; ----- Contour 2 -----
PTP {X 107.78, Y 86.02, Z 10.00, A 0, B 0, C 0}
LIN {X 107.78, Y 86.02, Z 0.00, A 0, B 0, C 0}
LIN {X 107.56, Y 86.02, Z 0.00, A 0, B 0, C 0} C_DIS
LIN {X 107.34, Y 86.02, Z 0.00, A 0, B 0, C 0} C_DIS
LIN {X 107.12, Y 86.02, Z 0.00, A 0, B 0, C 0} C_DIS
LIN {X 106.90, Y 86.02, Z 0.00, A 0, B 0, C 0} C_DIS
LIN {X 106.69, Y 86.03, Z 0.00, A 0, B 0, C 0} C_DIS
LIN {X 106.47, Y 86.03, Z 0.00, A 0, B 0, C 0} C_DIS
LIN {X 106.25, Y 86.04, Z 0.00, A 0, B 0, C 0} C_DIS
LIN {X 106.03, Y 86.04, Z 0.00, A 0, B 0, C 0} C_DIS
LIN {X 105.82, Y 86.04, Z 0.00, A 0, B 0, C 0} C_DIS
LIN {X 105.60, Y 86.03, Z 0.00, A 0, B 0, C 0} C_DIS
LIN {X 105.38, Y 86.02, Z 0.00, A 0, B 0, C 0} C_DIS
LIN {X 105.17, Y 86.00, Z 0.00, A 0, B 0, C 0} C_DIS
LIN {X 104.95, Y 85.97, Z 0.00, A 0, B 0, C 0} C_DIS
LIN {X 104.74, Y 85.94, Z 0.00, A 0, B 0, C 0} C_DIS
LIN {X 104.52, Y 85.90, Z 0.00, A 0, B 0, C 0} C_DIS
LIN {X 104.31, Y 85.85, Z 0.00, A 0, B 0, C 0} C_DIS
LIN {X 104.09, Y 85.79, Z 0.00, A 0, B 0, C 0} C_DIS
LIN {X 103.88, Y 85.73, Z 0.00, A 0, B 0, C 0} C_DIS
LIN {X 103.67, Y 85.67, Z 0.00, A 0, B 0, C 0} C_DIS
LIN {X 103.45, Y 85.60, Z 0.00, A 0, B 0, C 0} C_DIS
LIN {X 103.24, Y 85.53, Z 0.00, A 0, B 0, C 0} C_DIS
LIN {X 103.03, Y 85.46, Z 0.00, A 0, B 0, C 0} C_DIS
LIN {X 102.82, Y 85.39, Z 0.00, A 0, B 0, C 0} C_DIS
LIN {X 102.61, Y 85.31, Z 0.00, A 0, B 0, C 0} C_DIS
LIN {X 102.40, Y 85.24, Z 0.00, A 0, B 0, C 0} C_DIS
LIN {X 102.18, Y 85.17, Z 0.00, A 0, B 0, C 0} C_DIS
LIN {X 101.97, Y 85.09, Z 0.00, A 0, B 0, C 0} C_DIS
LIN {X 101.76, Y 85.01, Z 0.00, A 0, B 0, C 0} C_DIS
LIN {X 101.55, Y 84.94, Z 0.00, A 0, B 0, C 0} C_DIS
LIN {X 101.34, Y 84.85, Z 0.00, A 0, B 0, C 0} C_DIS
LIN {X 101.14, Y 84.77, Z 0.00, A 0, B 0, C 0} C_DIS
LIN {X 100.93, Y 84.68, Z 0.00, A 0, B 0, C 0} C_DIS
LIN {X 100.72, Y 84.58, Z 0.00, A 0, B 0, C 0} C_DIS
LIN {X 100.51, Y 84.48, Z 0.00, A 0, B 0, C 0} C_DIS
LIN {X 100.31, Y 84.38, Z 0.00, A 0, B 0, C 0} C_DIS
LIN {X 100.10, Y 84.27, Z 0.00, A 0, B 0, C 0} C_DIS
LIN {X 99.90, Y 84.15, Z 0.00, A 0, B 0, C 0} C_DIS
LIN {X 99.70, Y 84.02, Z 0.00, A 0, B 0, C 0} C_DIS
LIN {X 99.50, Y 83.89, Z 0.00, A 0, B 0, C 0} C_DIS
LIN {X 99.31, Y 83.74, Z 0.00, A 0, B 0, C 0} C_DIS
LIN {X 99.11, Y 83.59, Z 0.00, A 0, B 0, C 0} C_DIS
LIN {X 98.93, Y 83.43, Z 0.00, A 0, B 0, C 0} C_DIS
LIN {X 98.74, Y 83.26, Z 0.00, A 0, B 0, C 0} C_DIS
LIN {X 98.56, Y 83.08, Z 0.00, A 0, B 0, C 0} C_DIS
LIN {X 98.38, Y 82.89, Z 0.00, A 0, B 0, C 0} C_DIS
LIN {X 98.20, Y 82.72, Z 0.00, A 0, B 0, C 0} C_DIS
LIN {X 98.01, Y 82.56, Z 0.00, A 0, B 0, C 0} C_DIS
LIN {X 97.82, Y 82.41, Z 0.00, A 0, B 0, C 0} C_DIS
LIN {X 97.62, Y 82.28, Z 0.00, A 0, B 0, C 0} C_DIS
LIN {X 97.42, Y 82.13, Z 0.00, A 0, B 0, C 0} C_DIS
LIN {X 97.23, Y 81.97, Z 0.00, A 0, B 0, C 0} C_DIS
LIN {X 97.05, Y 81.80, Z 0.00, A 0, B 0, C 0} C_DIS
LIN {X 96.87, Y 81.61, Z 0.00, A 0, B 0, C 0} C_DIS
LIN {X 96.71, Y 81.40, Z 0.00, A 0, B 0, C 0} C_DIS
LIN {X 96.55, Y 81.17, Z 0.00, A 0, B 0, C 0} C_DIS
LIN {X 96.40, Y 80.93, Z 0.00, A 0, B 0, C 0} C_DIS
LIN {X 96.26, Y 80.69, Z 0.00, A 0, B 0, C 0} C_DIS
LIN {X 96.10, Y 80.45, Z 0.00, A 0, B 0, C 0} C_DIS
LIN {X 95.94, Y 80.23, Z 0.00, A 0, B 0, C 0} C_DIS
LIN {X 95.78, Y 80.01, Z 0.00, A 0, B 0, C 0} C_DIS
LIN {X 95.61, Y 79.81, Z 0.00, A 0, B 0, C 0} C_DIS
LIN {X 95.44, Y 79.60, Z 0.00, A 0, B 0, C 0} C_DIS
LIN {X 95.28, Y 79.39, Z 0.00, A 0, B 0, C 0} C_DIS
LIN {X 95.11, Y 79.18, Z 0.00, A 0, B 0, C 0} C_DIS
LIN {X 94.95, Y 78.96, Z 0.00, A 0, B 0, C 0} C_DIS
LIN {X 94.80, Y 78.73, Z 0.00, A 0, B 0, C 0} C_DIS
LIN {X 94.64, Y 78.51, Z 0.00, A 0, B 0, C 0} C_DIS
LIN {X 94.49, Y 78.27, Z 0.00, A 0, B 0, C 0} C_DIS
LIN {X 94.34, Y 78.04, Z 0.00, A 0, B 0, C 0} C_DIS
LIN {X 94.20, Y 77.80, Z 0.00, A 0, B 0, C 0} C_DIS
LIN {X 94.06, Y 77.55, Z 0.00, A 0, B 0, C 0} C_DIS
LIN {X 93.92, Y 77.31, Z 0.00, A 0, B 0, C 0} C_DIS
LIN {X 93.78, Y 77.05, Z 0.00, A 0, B 0, C 0} C_DIS
LIN {X 93.64, Y 76.80, Z 0.00, A 0, B 0, C 0} C_DIS
LIN {X 93.51, Y 76.54, Z 0.00, A 0, B 0, C 0} C_DIS
LIN {X 93.38, Y 76.28, Z 0.00, A 0, B 0, C 0} C_DIS
LIN {X 93.25, Y 76.01, Z 0.00, A 0, B 0, C 0} C_DIS
LIN {X 93.13, Y 75.74, Z 0.00, A 0, B 0, C 0} C_DIS
LIN {X 93.00, Y 75.47, Z 0.00, A 0, B 0, C 0} C_DIS
LIN {X 92.88, Y 75.20, Z 0.00, A 0, B 0, C 0} C_DIS
LIN {X 92.76, Y 74.93, Z 0.00, A 0, B 0, C 0} C_DIS
LIN {X 92.64, Y 74.65, Z 0.00, A 0, B 0, C 0} C_DIS
LIN {X 92.53, Y 74.38, Z 0.00, A 0, B 0, C 0} C_DIS
LIN {X 92.41, Y 74.10, Z 0.00, A 0, B 0, C 0} C_DIS
LIN {X 92.30, Y 73.82, Z 0.00, A 0, B 0, C 0} C_DIS
LIN {X 92.19, Y 73.54, Z 0.00, A 0, B 0, C 0} C_DIS
LIN {X 92.08, Y 73.26, Z 0.00, A 0, B 0, C 0} C_DIS
LIN {X 91.98, Y 72.97, Z 0.00, A 0, B 0, C 0} C_DIS
LIN {X 91.87, Y 72.69, Z 0.00, A 0, B 0, C 0} C_DIS
LIN {X 91.77, Y 72.40, Z 0.00, A 0, B 0, C 0} C_DIS
LIN {X 91.67, Y 72.11, Z 0.00, A 0, B 0, C 0} C_DIS
LIN {X 91.57, Y 71.82, Z 0.00, A 0, B 0, C 0} C_DIS
LIN {X 91.48, Y 71.52, Z 0.00, A 0, B 0, C 0} C_DIS
LIN {X 91.39, Y 71.23, Z 0.00, A 0, B 0, C 0} C_DIS
LIN {X 91.30, Y 70.93, Z 0.00, A 0, B 0, C 0} C_DIS
LIN {X 91.22, Y 70.63, Z 0.00, A 0, B 0, C 0} C_DIS
LIN {X 91.14, Y 70.32, Z 0.00, A 0, B 0, C 0} C_DIS
LIN {X 91.06, Y 70.02, Z 0.00, A 0, B 0, C 0} C_DIS
LIN {X 91.00, Y 69.71, Z 0.00, A 0, B 0, C 0} C_DIS
LIN {X 90.94, Y 69.39, Z 0.00, A 0, B 0, C 0} C_DIS
LIN {X 90.88, Y 69.08, Z 0.00, A 0, B 0, C 0} C_DIS
LIN {X 90.83, Y 68.76, Z 0.00, A 0, B 0, C 0} C_DIS
LIN {X 90.79, Y 68.44, Z 0.00, A 0, B 0, C 0} C_DIS
LIN {X 90.74, Y 68.12, Z 0.00, A 0, B 0, C 0} C_DIS
LIN {X 90.69, Y 67.80, Z 0.00, A 0, B 0, C 0} C_DIS
LIN {X 90.63, Y 67.48, Z 0.00, A 0, B 0, C 0} C_DIS
LIN {X 90.57, Y 67.17, Z 0.00, A 0, B 0, C 0} C_DIS
LIN {X 90.50, Y 66.86, Z 0.00, A 0, B 0, C 0} C_DIS
LIN {X 90.42, Y 66.56, Z 0.00, A 0, B 0, C 0} C_DIS
LIN {X 90.34, Y 66.25, Z 0.00, A 0, B 0, C 0} C_DIS
LIN {X 90.26, Y 65.94, Z 0.00, A 0, B 0, C 0} C_DIS
LIN {X 90.20, Y 65.63, Z 0.00, A 0, B 0, C 0} C_DIS
LIN {X 90.15, Y 65.31, Z 0.00, A 0, B 0, C 0} C_DIS
LIN {X 90.11, Y 64.99, Z 0.00, A 0, B 0, C 0} C_DIS
LIN {X 90.08, Y 64.67, Z 0.00, A 0, B 0, C 0} C_DIS
LIN {X 90.05, Y 64.34, Z 0.00, A 0, B 0, C 0} C_DIS
LIN {X 90.04, Y 64.01, Z 0.00, A 0, B 0, C 0} C_DIS
LIN {X 90.03, Y 63.69, Z 0.00, A 0, B 0, C 0} C_DIS
LIN {X 90.02, Y 63.36, Z 0.00, A 0, B 0, C 0} C_DIS
LIN {X 90.02, Y 63.03, Z 0.00, A 0, B 0, C 0} C_DIS
LIN {X 90.02, Y 62.70, Z 0.00, A 0, B 0, C 0} C_DIS
LIN {X 90.02, Y 62.38, Z 0.00, A 0, B 0, C 0} C_DIS
LIN {X 90.03, Y 62.05, Z 0.00, A 0, B 0, C 0} C_DIS
LIN {X 90.03, Y 61.72, Z 0.00, A 0, B 0, C 0} C_DIS
LIN {X 90.03, Y 61.39, Z 0.00, A 0, B 0, C 0} C_DIS
LIN {X 90.03, Y 61.07, Z 0.00, A 0, B 0, C 0} C_DIS
LIN {X 90.03, Y 60.74, Z 0.00, A 0, B 0, C 0} C_DIS
LIN {X 90.03, Y 60.41, Z 0.00, A 0, B 0, C 0} C_DIS
LIN {X 90.03, Y 60.08, Z 0.00, A 0, B 0, C 0} C_DIS
LIN {X 90.03, Y 59.76, Z 0.00, A 0, B 0, C 0} C_DIS
LIN {X 90.03, Y 59.43, Z 0.00, A 0, B 0, C 0} C_DIS
LIN {X 90.03, Y 59.10, Z 0.00, A 0, B 0, C 0} C_DIS
LIN {X 90.03, Y 58.77, Z 0.00, A 0, B 0, C 0} C_DIS
LIN {X 90.03, Y 58.44, Z 0.00, A 0, B 0, C 0} C_DIS
LIN {X 90.03, Y 58.12, Z 0.00, A 0, B 0, C 0} C_DIS
LIN {X 90.03, Y 57.79, Z 0.00, A 0, B 0, C 0} C_DIS
LIN {X 90.03, Y 57.46, Z 0.00, A 0, B 0, C 0} C_DIS
LIN {X 90.03, Y 57.13, Z 0.00, A 0, B 0, C 0} C_DIS
LIN {X 90.03, Y 56.80, Z 0.00, A 0, B 0, C 0} C_DIS
LIN {X 90.03, Y 56.48, Z 0.00, A 0, B 0, C 0} C_DIS
LIN {X 90.03, Y 56.15, Z 0.00, A 0, B 0, C 0} C_DIS
LIN {X 90.03, Y 55.82, Z 0.00, A 0, B 0, C 0} C_DIS
LIN {X 90.03, Y 55.49, Z 0.00, A 0, B 0, C 0} C_DIS
LIN {X 90.03, Y 55.17, Z 0.00, A 0, B 0, C 0} C_DIS
LIN {X 90.03, Y 54.84, Z 0.00, A 0, B 0, C 0} C_DIS
LIN {X 90.03, Y 54.51, Z 0.00, A 0, B 0, C 0} C_DIS
LIN {X 90.03, Y 54.18, Z 0.00, A 0, B 0, C 0} C_DIS
LIN {X 90.03, Y 53.86, Z 0.00, A 0, B 0, C 0} C_DIS
LIN {X 90.03, Y 53.53, Z 0.00, A 0, B 0, C 0} C_DIS
LIN {X 90.03, Y 53.20, Z 0.00, A 0, B 0, C 0} C_DIS
LIN {X 90.03, Y 52.87, Z 0.00, A 0, B 0, C 0} C_DIS
LIN {X 90.03, Y 52.55, Z 0.00, A 0, B 0, C 0} C_DIS
LIN {X 90.03, Y 52.22, Z 0.00, A 0, B 0, C 0} C_DIS
LIN {X 90.03, Y 51.89, Z 0.00, A 0, B 0, C 0} C_DIS
LIN {X 90.03, Y 51.56, Z 0.00, A 0, B 0, C 0} C_DIS
LIN {X 90.03, Y 51.24, Z 0.00, A 0, B 0, C 0} C_DIS
LIN {X 90.03, Y 50.91, Z 0.00, A 0, B 0, C 0} C_DIS
LIN {X 90.03, Y 50.58, Z 0.00, A 0, B 0, C 0} C_DIS
LIN {X 90.03, Y 50.25, Z 0.00, A 0, B 0, C 0} C_DIS
LIN {X 90.03, Y 49.92, Z 0.00, A 0, B 0, C 0} C_DIS
LIN {X 90.03, Y 49.60, Z 0.00, A 0, B 0, C 0} C_DIS
LIN {X 90.02, Y 49.27, Z 0.00, A 0, B 0, C 0} C_DIS
LIN {X 90.02, Y 48.94, Z 0.00, A 0, B 0, C 0} C_DIS
LIN {X 90.02, Y 48.61, Z 0.00, A 0, B 0, C 0} C_DIS
LIN {X 90.02, Y 48.28, Z 0.00, A 0, B 0, C 0} C_DIS
LIN {X 90.02, Y 47.95, Z 0.00, A 0, B 0, C 0} C_DIS
LIN {X 90.03, Y 47.62, Z 0.00, A 0, B 0, C 0} C_DIS
LIN {X 90.04, Y 47.30, Z 0.00, A 0, B 0, C 0} C_DIS
LIN {X 90.06, Y 46.97, Z 0.00, A 0, B 0, C 0} C_DIS
LIN {X 90.08, Y 46.65, Z 0.00, A 0, B 0, C 0} C_DIS
LIN {X 90.11, Y 46.33, Z 0.00, A 0, B 0, C 0} C_DIS
LIN {X 90.15, Y 46.01, Z 0.00, A 0, B 0, C 0} C_DIS
LIN {X 90.19, Y 45.69, Z 0.00, A 0, B 0, C 0} C_DIS
LIN {X 90.24, Y 45.37, Z 0.00, A 0, B 0, C 0} C_DIS
LIN {X 90.30, Y 45.06, Z 0.00, A 0, B 0, C 0} C_DIS
LIN {X 90.37, Y 44.75, Z 0.00, A 0, B 0, C 0} C_DIS
LIN {X 90.44, Y 44.44, Z 0.00, A 0, B 0, C 0} C_DIS
LIN {X 90.52, Y 44.13, Z 0.00, A 0, B 0, C 0} C_DIS
LIN {X 90.60, Y 43.83, Z 0.00, A 0, B 0, C 0} C_DIS
LIN {X 90.69, Y 43.53, Z 0.00, A 0, B 0, C 0} C_DIS
LIN {X 90.78, Y 43.23, Z 0.00, A 0, B 0, C 0} C_DIS
LIN {X 90.87, Y 42.93, Z 0.00, A 0, B 0, C 0} C_DIS
LIN {X 90.96, Y 42.63, Z 0.00, A 0, B 0, C 0} C_DIS
LIN {X 91.05, Y 42.34, Z 0.00, A 0, B 0, C 0} C_DIS
LIN {X 91.15, Y 42.04, Z 0.00, A 0, B 0, C 0} C_DIS
LIN {X 91.24, Y 41.75, Z 0.00, A 0, B 0, C 0} C_DIS
LIN {X 91.34, Y 41.46, Z 0.00, A 0, B 0, C 0} C_DIS
LIN {X 91.44, Y 41.17, Z 0.00, A 0, B 0, C 0} C_DIS
LIN {X 91.54, Y 40.89, Z 0.00, A 0, B 0, C 0} C_DIS
LIN {X 91.64, Y 40.60, Z 0.00, A 0, B 0, C 0} C_DIS
LIN {X 91.75, Y 40.32, Z 0.00, A 0, B 0, C 0} C_DIS
LIN {X 91.85, Y 40.03, Z 0.00, A 0, B 0, C 0} C_DIS
LIN {X 91.96, Y 39.75, Z 0.00, A 0, B 0, C 0} C_DIS
LIN {X 92.08, Y 39.47, Z 0.00, A 0, B 0, C 0} C_DIS
LIN {X 92.19, Y 39.19, Z 0.00, A 0, B 0, C 0} C_DIS
LIN {X 92.31, Y 38.92, Z 0.00, A 0, B 0, C 0} C_DIS
LIN {X 92.43, Y 38.64, Z 0.00, A 0, B 0, C 0} C_DIS
LIN {X 92.55, Y 38.37, Z 0.00, A 0, B 0, C 0} C_DIS
LIN {X 92.68, Y 38.11, Z 0.00, A 0, B 0, C 0} C_DIS
LIN {X 92.81, Y 37.84, Z 0.00, A 0, B 0, C 0} C_DIS
LIN {X 92.94, Y 37.59, Z 0.00, A 0, B 0, C 0} C_DIS
LIN {X 93.08, Y 37.33, Z 0.00, A 0, B 0, C 0} C_DIS
LIN {X 93.22, Y 37.08, Z 0.00, A 0, B 0, C 0} C_DIS
LIN {X 93.37, Y 36.84, Z 0.00, A 0, B 0, C 0} C_DIS
LIN {X 93.51, Y 36.60, Z 0.00, A 0, B 0, C 0} C_DIS
LIN {X 93.66, Y 36.36, Z 0.00, A 0, B 0, C 0} C_DIS
LIN {X 93.81, Y 36.12, Z 0.00, A 0, B 0, C 0} C_DIS
LIN {X 93.97, Y 35.89, Z 0.00, A 0, B 0, C 0} C_DIS
LIN {X 94.12, Y 35.66, Z 0.00, A 0, B 0, C 0} C_DIS
LIN {X 94.27, Y 35.43, Z 0.00, A 0, B 0, C 0} C_DIS
LIN {X 94.43, Y 35.20, Z 0.00, A 0, B 0, C 0} C_DIS
LIN {X 94.58, Y 34.97, Z 0.00, A 0, B 0, C 0} C_DIS
LIN {X 94.74, Y 34.74, Z 0.00, A 0, B 0, C 0} C_DIS
LIN {X 94.89, Y 34.51, Z 0.00, A 0, B 0, C 0} C_DIS
LIN {X 95.05, Y 34.28, Z 0.00, A 0, B 0, C 0} C_DIS
LIN {X 95.20, Y 34.05, Z 0.00, A 0, B 0, C 0} C_DIS
LIN {X 95.35, Y 33.82, Z 0.00, A 0, B 0, C 0} C_DIS
LIN {X 95.51, Y 33.58, Z 0.00, A 0, B 0, C 0} C_DIS
LIN {X 95.66, Y 33.35, Z 0.00, A 0, B 0, C 0} C_DIS
LIN {X 95.82, Y 33.12, Z 0.00, A 0, B 0, C 0} C_DIS
LIN {X 95.97, Y 32.89, Z 0.00, A 0, B 0, C 0} C_DIS
LIN {X 96.13, Y 32.66, Z 0.00, A 0, B 0, C 0} C_DIS
LIN {X 96.28, Y 32.43, Z 0.00, A 0, B 0, C 0} C_DIS
LIN {X 96.43, Y 32.20, Z 0.00, A 0, B 0, C 0} C_DIS
LIN {X 96.59, Y 31.97, Z 0.00, A 0, B 0, C 0} C_DIS
LIN {X 96.74, Y 31.73, Z 0.00, A 0, B 0, C 0} C_DIS
LIN {X 96.90, Y 31.50, Z 0.00, A 0, B 0, C 0} C_DIS
LIN {X 97.05, Y 31.27, Z 0.00, A 0, B 0, C 0} C_DIS
LIN {X 97.20, Y 31.04, Z 0.00, A 0, B 0, C 0} C_DIS
LIN {X 97.36, Y 30.81, Z 0.00, A 0, B 0, C 0} C_DIS
LIN {X 97.51, Y 30.58, Z 0.00, A 0, B 0, C 0} C_DIS
LIN {X 97.66, Y 30.34, Z 0.00, A 0, B 0, C 0} C_DIS
LIN {X 97.82, Y 30.11, Z 0.00, A 0, B 0, C 0} C_DIS
LIN {X 97.97, Y 29.88, Z 0.00, A 0, B 0, C 0} C_DIS
LIN {X 98.13, Y 29.65, Z 0.00, A 0, B 0, C 0} C_DIS
LIN {X 98.28, Y 29.42, Z 0.00, A 0, B 0, C 0} C_DIS
LIN {X 98.43, Y 29.18, Z 0.00, A 0, B 0, C 0} C_DIS
LIN {X 98.59, Y 28.95, Z 0.00, A 0, B 0, C 0} C_DIS
LIN {X 98.74, Y 28.72, Z 0.00, A 0, B 0, C 0} C_DIS
LIN {X 98.89, Y 28.49, Z 0.00, A 0, B 0, C 0} C_DIS
LIN {X 99.05, Y 28.26, Z 0.00, A 0, B 0, C 0} C_DIS
LIN {X 99.20, Y 28.03, Z 0.00, A 0, B 0, C 0} C_DIS
LIN {X 99.35, Y 27.79, Z 0.00, A 0, B 0, C 0} C_DIS
LIN {X 99.51, Y 27.56, Z 0.00, A 0, B 0, C 0} C_DIS
LIN {X 99.66, Y 27.33, Z 0.00, A 0, B 0, C 0} C_DIS
LIN {X 99.82, Y 27.10, Z 0.00, A 0, B 0, C 0} C_DIS
LIN {X 99.97, Y 26.87, Z 0.00, A 0, B 0, C 0} C_DIS
LIN {X 100.12, Y 26.63, Z 0.00, A 0, B 0, C 0} C_DIS
LIN {X 100.28, Y 26.40, Z 0.00, A 0, B 0, C 0} C_DIS
LIN {X 100.43, Y 26.17, Z 0.00, A 0, B 0, C 0} C_DIS
LIN {X 100.58, Y 25.94, Z 0.00, A 0, B 0, C 0} C_DIS
LIN {X 100.74, Y 25.71, Z 0.00, A 0, B 0, C 0} C_DIS
LIN {X 100.89, Y 25.47, Z 0.00, A 0, B 0, C 0} C_DIS
LIN {X 101.05, Y 25.24, Z 0.00, A 0, B 0, C 0} C_DIS
LIN {X 101.20, Y 25.01, Z 0.00, A 0, B 0, C 0} C_DIS
LIN {X 101.35, Y 24.78, Z 0.00, A 0, B 0, C 0} C_DIS
LIN {X 101.51, Y 24.55, Z 0.00, A 0, B 0, C 0} C_DIS
LIN {X 101.66, Y 24.31, Z 0.00, A 0, B 0, C 0} C_DIS
LIN {X 101.81, Y 24.08, Z 0.00, A 0, B 0, C 0} C_DIS
LIN {X 101.97, Y 23.85, Z 0.00, A 0, B 0, C 0} C_DIS
LIN {X 102.12, Y 23.62, Z 0.00, A 0, B 0, C 0} C_DIS
LIN {X 102.28, Y 23.39, Z 0.00, A 0, B 0, C 0} C_DIS
LIN {X 102.43, Y 23.16, Z 0.00, A 0, B 0, C 0} C_DIS
LIN {X 102.58, Y 22.92, Z 0.00, A 0, B 0, C 0} C_DIS
LIN {X 102.74, Y 22.69, Z 0.00, A 0, B 0, C 0} C_DIS
LIN {X 102.89, Y 22.46, Z 0.00, A 0, B 0, C 0} C_DIS
LIN {X 103.04, Y 22.23, Z 0.00, A 0, B 0, C 0} C_DIS
LIN {X 103.20, Y 22.00, Z 0.00, A 0, B 0, C 0} C_DIS
LIN {X 103.35, Y 21.77, Z 0.00, A 0, B 0, C 0} C_DIS
LIN {X 103.51, Y 21.53, Z 0.00, A 0, B 0, C 0} C_DIS
LIN {X 103.66, Y 21.30, Z 0.00, A 0, B 0, C 0} C_DIS
LIN {X 103.81, Y 21.07, Z 0.00, A 0, B 0, C 0} C_DIS
LIN {X 103.97, Y 20.84, Z 0.00, A 0, B 0, C 0} C_DIS
LIN {X 104.12, Y 20.61, Z 0.00, A 0, B 0, C 0} C_DIS
LIN {X 104.27, Y 20.38, Z 0.00, A 0, B 0, C 0} C_DIS
LIN {X 104.43, Y 20.14, Z 0.00, A 0, B 0, C 0} C_DIS
LIN {X 104.58, Y 19.91, Z 0.00, A 0, B 0, C 0} C_DIS
LIN {X 104.74, Y 19.68, Z 0.00, A 0, B 0, C 0} C_DIS
LIN {X 104.89, Y 19.45, Z 0.00, A 0, B 0, C 0} C_DIS
LIN {X 105.04, Y 19.22, Z 0.00, A 0, B 0, C 0} C_DIS
LIN {X 105.20, Y 18.99, Z 0.00, A 0, B 0, C 0} C_DIS
LIN {X 105.35, Y 18.75, Z 0.00, A 0, B 0, C 0} C_DIS
LIN {X 105.50, Y 18.52, Z 0.00, A 0, B 0, C 0} C_DIS
LIN {X 105.66, Y 18.29, Z 0.00, A 0, B 0, C 0} C_DIS
LIN {X 105.81, Y 18.06, Z 0.00, A 0, B 0, C 0} C_DIS
LIN {X 105.97, Y 17.83, Z 0.00, A 0, B 0, C 0} C_DIS
LIN {X 106.12, Y 17.60, Z 0.00, A 0, B 0, C 0} C_DIS
LIN {X 106.27, Y 17.36, Z 0.00, A 0, B 0, C 0} C_DIS
LIN {X 106.43, Y 17.13, Z 0.00, A 0, B 0, C 0} C_DIS
LIN {X 106.58, Y 16.90, Z 0.00, A 0, B 0, C 0} C_DIS
LIN {X 106.74, Y 16.67, Z 0.00, A 0, B 0, C 0} C_DIS
LIN {X 106.89, Y 16.44, Z 0.00, A 0, B 0, C 0} C_DIS
LIN {X 107.04, Y 16.21, Z 0.00, A 0, B 0, C 0} C_DIS
LIN {X 107.20, Y 15.97, Z 0.00, A 0, B 0, C 0} C_DIS
LIN {X 107.35, Y 15.74, Z 0.00, A 0, B 0, C 0} C_DIS
LIN {X 107.50, Y 15.51, Z 0.00, A 0, B 0, C 0} C_DIS
LIN {X 107.66, Y 15.28, Z 0.00, A 0, B 0, C 0} C_DIS
LIN {X 107.81, Y 15.05, Z 0.00, A 0, B 0, C 0} C_DIS
LIN {X 107.97, Y 14.82, Z 0.00, A 0, B 0, C 0} C_DIS
LIN {X 108.12, Y 14.58, Z 0.00, A 0, B 0, C 0} C_DIS
LIN {X 108.27, Y 14.35, Z 0.00, A 0, B 0, C 0} C_DIS
LIN {X 108.43, Y 14.12, Z 0.00, A 0, B 0, C 0} C_DIS
LIN {X 108.58, Y 13.89, Z 0.00, A 0, B 0, C 0} C_DIS
LIN {X 108.73, Y 13.66, Z 0.00, A 0, B 0, C 0} C_DIS
LIN {X 108.89, Y 13.43, Z 0.00, A 0, B 0, C 0} C_DIS
LIN {X 109.04, Y 13.19, Z 0.00, A 0, B 0, C 0} C_DIS
LIN {X 109.20, Y 12.96, Z 0.00, A 0, B 0, C 0} C_DIS
LIN {X 109.35, Y 12.73, Z 0.00, A 0, B 0, C 0} C_DIS
LIN {X 109.50, Y 12.50, Z 0.00, A 0, B 0, C 0} C_DIS
LIN {X 109.66, Y 12.27, Z 0.00, A 0, B 0, C 0} C_DIS
LIN {X 109.81, Y 12.03, Z 0.00, A 0, B 0, C 0} C_DIS
LIN {X 109.96, Y 11.80, Z 0.00, A 0, B 0, C 0} C_DIS
LIN {X 110.12, Y 11.57, Z 0.00, A 0, B 0, C 0} C_DIS
LIN {X 110.27, Y 11.34, Z 0.00, A 0, B 0, C 0} C_DIS
LIN {X 110.43, Y 11.11, Z 0.00, A 0, B 0, C 0} C_DIS
LIN {X 110.58, Y 10.88, Z 0.00, A 0, B 0, C 0} C_DIS
LIN {X 110.73, Y 10.64, Z 0.00, A 0, B 0, C 0} C_DIS
LIN {X 110.89, Y 10.41, Z 0.00, A 0, B 0, C 0} C_DIS
LIN {X 111.04, Y 10.18, Z 0.00, A 0, B 0, C 0} C_DIS
LIN {X 111.19, Y 9.95, Z 0.00, A 0, B 0, C 0} C_DIS
LIN {X 111.35, Y 9.72, Z 0.00, A 0, B 0, C 0} C_DIS
LIN {X 111.50, Y 9.48, Z 0.00, A 0, B 0, C 0} C_DIS
LIN {X 111.66, Y 9.25, Z 0.00, A 0, B 0, C 0} C_DIS
LIN {X 111.81, Y 9.02, Z 0.00, A 0, B 0, C 0} C_DIS
LIN {X 111.96, Y 8.79, Z 0.00, A 0, B 0, C 0} C_DIS
LIN {X 112.12, Y 8.56, Z 0.00, A 0, B 0, C 0} C_DIS
LIN {X 112.27, Y 8.32, Z 0.00, A 0, B 0, C 0} C_DIS
LIN {X 112.42, Y 8.09, Z 0.00, A 0, B 0, C 0} C_DIS
LIN {X 112.58, Y 7.86, Z 0.00, A 0, B 0, C 0} C_DIS
LIN {X 112.73, Y 7.62, Z 0.00, A 0, B 0, C 0} C_DIS
LIN {X 112.88, Y 7.39, Z 0.00, A 0, B 0, C 0} C_DIS
LIN {X 113.04, Y 7.16, Z 0.00, A 0, B 0, C 0} C_DIS
LIN {X 113.19, Y 6.93, Z 0.00, A 0, B 0, C 0} C_DIS
LIN {X 113.35, Y 6.71, Z 0.00, A 0, B 0, C 0} C_DIS
LIN {X 113.51, Y 6.49, Z 0.00, A 0, B 0, C 0} C_DIS
LIN {X 113.67, Y 6.27, Z 0.00, A 0, B 0, C 0} C_DIS
LIN {X 113.84, Y 6.06, Z 0.00, A 0, B 0, C 0} C_DIS
LIN {X 114.01, Y 5.86, Z 0.00, A 0, B 0, C 0} C_DIS
LIN {X 114.18, Y 5.67, Z 0.00, A 0, B 0, C 0} C_DIS
LIN {X 114.36, Y 5.48, Z 0.00, A 0, B 0, C 0} C_DIS
LIN {X 114.54, Y 5.29, Z 0.00, A 0, B 0, C 0} C_DIS
LIN {X 114.72, Y 5.12, Z 0.00, A 0, B 0, C 0} C_DIS
LIN {X 114.90, Y 4.94, Z 0.00, A 0, B 0, C 0} C_DIS
LIN {X 115.09, Y 4.76, Z 0.00, A 0, B 0, C 0} C_DIS
LIN {X 115.27, Y 4.59, Z 0.00, A 0, B 0, C 0} C_DIS
LIN {X 115.46, Y 4.41, Z 0.00, A 0, B 0, C 0} C_DIS
LIN {X 115.64, Y 4.24, Z 0.00, A 0, B 0, C 0} C_DIS
LIN {X 115.82, Y 4.05, Z 0.00, A 0, B 0, C 0} C_DIS
LIN {X 116.00, Y 3.87, Z 0.00, A 0, B 0, C 0} C_DIS
LIN {X 116.18, Y 3.68, Z 0.00, A 0, B 0, C 0} C_DIS
LIN {X 116.36, Y 3.49, Z 0.00, A 0, B 0, C 0} C_DIS
LIN {X 116.54, Y 3.31, Z 0.00, A 0, B 0, C 0} C_DIS
LIN {X 116.72, Y 3.13, Z 0.00, A 0, B 0, C 0} C_DIS
LIN {X 116.90, Y 2.96, Z 0.00, A 0, B 0, C 0} C_DIS
LIN {X 117.09, Y 2.80, Z 0.00, A 0, B 0, C 0} C_DIS
LIN {X 117.28, Y 2.65, Z 0.00, A 0, B 0, C 0} C_DIS
LIN {X 117.48, Y 2.52, Z 0.00, A 0, B 0, C 0} C_DIS
LIN {X 117.68, Y 2.41, Z 0.00, A 0, B 0, C 0} C_DIS
LIN {X 117.89, Y 2.30, Z 0.00, A 0, B 0, C 0} C_DIS
LIN {X 118.10, Y 2.21, Z 0.00, A 0, B 0, C 0} C_DIS
LIN {X 118.31, Y 2.10, Z 0.00, A 0, B 0, C 0} C_DIS
LIN {X 118.51, Y 2.00, Z 0.00, A 0, B 0, C 0} C_DIS
LIN {X 118.72, Y 1.88, Z 0.00, A 0, B 0, C 0} C_DIS
LIN {X 118.91, Y 1.75, Z 0.00, A 0, B 0, C 0} C_DIS
LIN {X 119.11, Y 1.61, Z 0.00, A 0, B 0, C 0} C_DIS
LIN {X 119.30, Y 1.47, Z 0.00, A 0, B 0, C 0} C_DIS
LIN {X 119.50, Y 1.34, Z 0.00, A 0, B 0, C 0} C_DIS
LIN {X 119.70, Y 1.22, Z 0.00, A 0, B 0, C 0} C_DIS
LIN {X 119.91, Y 1.13, Z 0.00, A 0, B 0, C 0} C_DIS
LIN {X 120.11, Y 1.05, Z 0.00, A 0, B 0, C 0} C_DIS
LIN {X 120.32, Y 0.99, Z 0.00, A 0, B 0, C 0} C_DIS
LIN {X 120.54, Y 0.93, Z 0.00, A 0, B 0, C 0} C_DIS
LIN {X 120.75, Y 0.88, Z 0.00, A 0, B 0, C 0} C_DIS
LIN {X 120.97, Y 0.83, Z 0.00, A 0, B 0, C 0} C_DIS
LIN {X 121.19, Y 0.79, Z 0.00, A 0, B 0, C 0} C_DIS
LIN {X 121.41, Y 0.73, Z 0.00, A 0, B 0, C 0} C_DIS
LIN {X 121.63, Y 0.68, Z 0.00, A 0, B 0, C 0} C_DIS
LIN {X 121.85, Y 0.61, Z 0.00, A 0, B 0, C 0} C_DIS
LIN {X 122.06, Y 0.56, Z 0.00, A 0, B 0, C 0} C_DIS
LIN {X 122.24, Y 0.61, Z 0.00, A 0, B 0, C 0} C_DIS
LIN {X 122.38, Y 0.80, Z 0.00, A 0, B 0, C 0} C_DIS
LIN {X 122.46, Y 1.10, Z 0.00, A 0, B 0, C 0} C_DIS
LIN {X 122.52, Y 1.43, Z 0.00, A 0, B 0, C 0} C_DIS
LIN {X 122.56, Y 1.76, Z 0.00, A 0, B 0, C 0} C_DIS
LIN {X 122.58, Y 2.09, Z 0.00, A 0, B 0, C 0} C_DIS
LIN {X 122.59, Y 2.42, Z 0.00, A 0, B 0, C 0} C_DIS
LIN {X 122.59, Y 2.75, Z 0.00, A 0, B 0, C 0} C_DIS
LIN {X 122.58, Y 3.08, Z 0.00, A 0, B 0, C 0} C_DIS
LIN {X 122.58, Y 3.41, Z 0.00, A 0, B 0, C 0} C_DIS
LIN {X 122.57, Y 3.73, Z 0.00, A 0, B 0, C 0} C_DIS
LIN {X 122.57, Y 4.06, Z 0.00, A 0, B 0, C 0} C_DIS
LIN {X 122.56, Y 4.39, Z 0.00, A 0, B 0, C 0} C_DIS
LIN {X 122.56, Y 4.72, Z 0.00, A 0, B 0, C 0} C_DIS
LIN {X 122.56, Y 5.05, Z 0.00, A 0, B 0, C 0} C_DIS
LIN {X 122.56, Y 5.38, Z 0.00, A 0, B 0, C 0} C_DIS
LIN {X 122.56, Y 5.70, Z 0.00, A 0, B 0, C 0} C_DIS
LIN {X 122.56, Y 6.03, Z 0.00, A 0, B 0, C 0} C_DIS
LIN {X 122.56, Y 6.36, Z 0.00, A 0, B 0, C 0} C_DIS
LIN {X 122.56, Y 6.69, Z 0.00, A 0, B 0, C 0} C_DIS
LIN {X 122.56, Y 7.01, Z 0.00, A 0, B 0, C 0} C_DIS
LIN {X 122.56, Y 7.34, Z 0.00, A 0, B 0, C 0} C_DIS
LIN {X 122.56, Y 7.67, Z 0.00, A 0, B 0, C 0} C_DIS
LIN {X 122.56, Y 8.00, Z 0.00, A 0, B 0, C 0} C_DIS
LIN {X 122.56, Y 8.32, Z 0.00, A 0, B 0, C 0} C_DIS
LIN {X 122.56, Y 8.65, Z 0.00, A 0, B 0, C 0} C_DIS
LIN {X 122.56, Y 8.98, Z 0.00, A 0, B 0, C 0} C_DIS
LIN {X 122.56, Y 9.31, Z 0.00, A 0, B 0, C 0} C_DIS
LIN {X 122.56, Y 9.64, Z 0.00, A 0, B 0, C 0} C_DIS
LIN {X 122.56, Y 9.96, Z 0.00, A 0, B 0, C 0} C_DIS
LIN {X 122.56, Y 10.29, Z 0.00, A 0, B 0, C 0} C_DIS
LIN {X 122.56, Y 10.62, Z 0.00, A 0, B 0, C 0} C_DIS
LIN {X 122.56, Y 10.95, Z 0.00, A 0, B 0, C 0} C_DIS
LIN {X 122.56, Y 11.27, Z 0.00, A 0, B 0, C 0} C_DIS
LIN {X 122.56, Y 11.60, Z 0.00, A 0, B 0, C 0} C_DIS
LIN {X 122.56, Y 11.93, Z 0.00, A 0, B 0, C 0} C_DIS
LIN {X 122.56, Y 12.26, Z 0.00, A 0, B 0, C 0} C_DIS
LIN {X 122.56, Y 12.58, Z 0.00, A 0, B 0, C 0} C_DIS
LIN {X 122.56, Y 12.91, Z 0.00, A 0, B 0, C 0} C_DIS
LIN {X 122.56, Y 13.24, Z 0.00, A 0, B 0, C 0} C_DIS
LIN {X 122.56, Y 13.57, Z 0.00, A 0, B 0, C 0} C_DIS
LIN {X 122.56, Y 13.90, Z 0.00, A 0, B 0, C 0} C_DIS
LIN {X 122.56, Y 14.22, Z 0.00, A 0, B 0, C 0} C_DIS
LIN {X 122.56, Y 14.55, Z 0.00, A 0, B 0, C 0} C_DIS
LIN {X 122.56, Y 14.88, Z 0.00, A 0, B 0, C 0} C_DIS
LIN {X 122.56, Y 15.21, Z 0.00, A 0, B 0, C 0} C_DIS
LIN {X 122.56, Y 15.53, Z 0.00, A 0, B 0, C 0} C_DIS
LIN {X 122.56, Y 15.86, Z 0.00, A 0, B 0, C 0} C_DIS
LIN {X 122.56, Y 16.19, Z 0.00, A 0, B 0, C 0} C_DIS
LIN {X 122.56, Y 16.52, Z 0.00, A 0, B 0, C 0} C_DIS
LIN {X 122.56, Y 16.84, Z 0.00, A 0, B 0, C 0} C_DIS
LIN {X 122.56, Y 17.17, Z 0.00, A 0, B 0, C 0} C_DIS
LIN {X 122.56, Y 17.50, Z 0.00, A 0, B 0, C 0} C_DIS
LIN {X 122.56, Y 17.83, Z 0.00, A 0, B 0, C 0} C_DIS
LIN {X 122.56, Y 18.16, Z 0.00, A 0, B 0, C 0} C_DIS
LIN {X 122.56, Y 18.48, Z 0.00, A 0, B 0, C 0} C_DIS
LIN {X 122.56, Y 18.81, Z 0.00, A 0, B 0, C 0} C_DIS
LIN {X 122.56, Y 19.14, Z 0.00, A 0, B 0, C 0} C_DIS
LIN {X 122.56, Y 19.47, Z 0.00, A 0, B 0, C 0} C_DIS
LIN {X 122.56, Y 19.79, Z 0.00, A 0, B 0, C 0} C_DIS
LIN {X 122.56, Y 20.12, Z 0.00, A 0, B 0, C 0} C_DIS
LIN {X 122.56, Y 20.45, Z 0.00, A 0, B 0, C 0} C_DIS
LIN {X 122.56, Y 20.78, Z 0.00, A 0, B 0, C 0} C_DIS
LIN {X 122.56, Y 21.10, Z 0.00, A 0, B 0, C 0} C_DIS
LIN {X 122.56, Y 21.43, Z 0.00, A 0, B 0, C 0} C_DIS
LIN {X 122.56, Y 21.76, Z 0.00, A 0, B 0, C 0} C_DIS
LIN {X 122.56, Y 22.09, Z 0.00, A 0, B 0, C 0} C_DIS
LIN {X 122.56, Y 22.42, Z 0.00, A 0, B 0, C 0} C_DIS
LIN {X 122.56, Y 22.74, Z 0.00, A 0, B 0, C 0} C_DIS
LIN {X 122.56, Y 23.07, Z 0.00, A 0, B 0, C 0} C_DIS
LIN {X 122.56, Y 23.40, Z 0.00, A 0, B 0, C 0} C_DIS
LIN {X 122.56, Y 23.73, Z 0.00, A 0, B 0, C 0} C_DIS
LIN {X 122.56, Y 24.05, Z 0.00, A 0, B 0, C 0} C_DIS
LIN {X 122.56, Y 24.38, Z 0.00, A 0, B 0, C 0} C_DIS
LIN {X 122.56, Y 24.71, Z 0.00, A 0, B 0, C 0} C_DIS
LIN {X 122.56, Y 25.04, Z 0.00, A 0, B 0, C 0} C_DIS
LIN {X 122.56, Y 25.37, Z 0.00, A 0, B 0, C 0} C_DIS
LIN {X 122.56, Y 25.69, Z 0.00, A 0, B 0, C 0} C_DIS
LIN {X 122.56, Y 26.02, Z 0.00, A 0, B 0, C 0} C_DIS
LIN {X 122.56, Y 26.35, Z 0.00, A 0, B 0, C 0} C_DIS
LIN {X 122.56, Y 26.68, Z 0.00, A 0, B 0, C 0} C_DIS
LIN {X 122.56, Y 27.00, Z 0.00, A 0, B 0, C 0} C_DIS
LIN {X 122.56, Y 27.33, Z 0.00, A 0, B 0, C 0} C_DIS
LIN {X 122.56, Y 27.66, Z 0.00, A 0, B 0, C 0} C_DIS
LIN {X 122.56, Y 27.99, Z 0.00, A 0, B 0, C 0} C_DIS
LIN {X 122.56, Y 28.31, Z 0.00, A 0, B 0, C 0} C_DIS
LIN {X 122.56, Y 28.64, Z 0.00, A 0, B 0, C 0} C_DIS
LIN {X 122.56, Y 28.97, Z 0.00, A 0, B 0, C 0} C_DIS
LIN {X 122.56, Y 29.30, Z 0.00, A 0, B 0, C 0} C_DIS
LIN {X 122.56, Y 29.63, Z 0.00, A 0, B 0, C 0} C_DIS
LIN {X 122.56, Y 29.95, Z 0.00, A 0, B 0, C 0} C_DIS
LIN {X 122.56, Y 30.28, Z 0.00, A 0, B 0, C 0} C_DIS
LIN {X 122.56, Y 30.61, Z 0.00, A 0, B 0, C 0} C_DIS
LIN {X 122.56, Y 30.94, Z 0.00, A 0, B 0, C 0} C_DIS
LIN {X 122.56, Y 31.26, Z 0.00, A 0, B 0, C 0} C_DIS
LIN {X 122.56, Y 31.59, Z 0.00, A 0, B 0, C 0} C_DIS
LIN {X 122.56, Y 31.92, Z 0.00, A 0, B 0, C 0} C_DIS
LIN {X 122.56, Y 32.25, Z 0.00, A 0, B 0, C 0} C_DIS
LIN {X 122.56, Y 32.58, Z 0.00, A 0, B 0, C 0} C_DIS
LIN {X 122.56, Y 32.90, Z 0.00, A 0, B 0, C 0} C_DIS
LIN {X 122.56, Y 33.23, Z 0.00, A 0, B 0, C 0} C_DIS
LIN {X 122.56, Y 33.56, Z 0.00, A 0, B 0, C 0} C_DIS
LIN {X 122.56, Y 33.89, Z 0.00, A 0, B 0, C 0} C_DIS
LIN {X 122.56, Y 34.21, Z 0.00, A 0, B 0, C 0} C_DIS
LIN {X 122.56, Y 34.54, Z 0.00, A 0, B 0, C 0} C_DIS
LIN {X 122.56, Y 34.87, Z 0.00, A 0, B 0, C 0} C_DIS
LIN {X 122.56, Y 35.20, Z 0.00, A 0, B 0, C 0} C_DIS
LIN {X 122.56, Y 35.53, Z 0.00, A 0, B 0, C 0} C_DIS
LIN {X 122.56, Y 35.85, Z 0.00, A 0, B 0, C 0} C_DIS
LIN {X 122.56, Y 36.18, Z 0.00, A 0, B 0, C 0} C_DIS
LIN {X 122.56, Y 36.51, Z 0.00, A 0, B 0, C 0} C_DIS
LIN {X 122.56, Y 36.84, Z 0.00, A 0, B 0, C 0} C_DIS
LIN {X 122.56, Y 37.16, Z 0.00, A 0, B 0, C 0} C_DIS
LIN {X 122.56, Y 37.49, Z 0.00, A 0, B 0, C 0} C_DIS
LIN {X 122.56, Y 37.82, Z 0.00, A 0, B 0, C 0} C_DIS
LIN {X 122.56, Y 38.15, Z 0.00, A 0, B 0, C 0} C_DIS
LIN {X 122.56, Y 38.47, Z 0.00, A 0, B 0, C 0} C_DIS
LIN {X 122.56, Y 38.80, Z 0.00, A 0, B 0, C 0} C_DIS
LIN {X 122.56, Y 39.13, Z 0.00, A 0, B 0, C 0} C_DIS
LIN {X 122.56, Y 39.46, Z 0.00, A 0, B 0, C 0} C_DIS
LIN {X 122.56, Y 39.79, Z 0.00, A 0, B 0, C 0} C_DIS
LIN {X 122.56, Y 40.11, Z 0.00, A 0, B 0, C 0} C_DIS
LIN {X 122.56, Y 40.44, Z 0.00, A 0, B 0, C 0} C_DIS
LIN {X 122.56, Y 40.77, Z 0.00, A 0, B 0, C 0} C_DIS
LIN {X 122.56, Y 41.10, Z 0.00, A 0, B 0, C 0} C_DIS
LIN {X 122.56, Y 41.42, Z 0.00, A 0, B 0, C 0} C_DIS
LIN {X 122.56, Y 41.75, Z 0.00, A 0, B 0, C 0} C_DIS
LIN {X 122.56, Y 42.08, Z 0.00, A 0, B 0, C 0} C_DIS
LIN {X 122.56, Y 42.41, Z 0.00, A 0, B 0, C 0} C_DIS
LIN {X 122.56, Y 42.74, Z 0.00, A 0, B 0, C 0} C_DIS
LIN {X 122.56, Y 43.06, Z 0.00, A 0, B 0, C 0} C_DIS
LIN {X 122.56, Y 43.39, Z 0.00, A 0, B 0, C 0} C_DIS
LIN {X 122.56, Y 43.72, Z 0.00, A 0, B 0, C 0} C_DIS
LIN {X 122.56, Y 44.05, Z 0.00, A 0, B 0, C 0} C_DIS
LIN {X 122.56, Y 44.37, Z 0.00, A 0, B 0, C 0} C_DIS
LIN {X 122.56, Y 44.70, Z 0.00, A 0, B 0, C 0} C_DIS
LIN {X 122.56, Y 45.03, Z 0.00, A 0, B 0, C 0} C_DIS
LIN {X 122.56, Y 45.36, Z 0.00, A 0, B 0, C 0} C_DIS
LIN {X 122.56, Y 45.69, Z 0.00, A 0, B 0, C 0} C_DIS
LIN {X 122.56, Y 46.01, Z 0.00, A 0, B 0, C 0} C_DIS
LIN {X 122.56, Y 46.34, Z 0.00, A 0, B 0, C 0} C_DIS
LIN {X 122.56, Y 46.67, Z 0.00, A 0, B 0, C 0} C_DIS
LIN {X 122.56, Y 47.00, Z 0.00, A 0, B 0, C 0} C_DIS
LIN {X 122.56, Y 47.32, Z 0.00, A 0, B 0, C 0} C_DIS
LIN {X 122.56, Y 47.65, Z 0.00, A 0, B 0, C 0} C_DIS
LIN {X 122.56, Y 47.98, Z 0.00, A 0, B 0, C 0} C_DIS
LIN {X 122.56, Y 48.31, Z 0.00, A 0, B 0, C 0} C_DIS
LIN {X 122.56, Y 48.63, Z 0.00, A 0, B 0, C 0} C_DIS
LIN {X 122.56, Y 48.96, Z 0.00, A 0, B 0, C 0} C_DIS
LIN {X 122.56, Y 49.29, Z 0.00, A 0, B 0, C 0} C_DIS
LIN {X 122.56, Y 49.62, Z 0.00, A 0, B 0, C 0} C_DIS
LIN {X 122.56, Y 49.95, Z 0.00, A 0, B 0, C 0} C_DIS
LIN {X 122.56, Y 50.27, Z 0.00, A 0, B 0, C 0} C_DIS
LIN {X 122.56, Y 50.60, Z 0.00, A 0, B 0, C 0} C_DIS
LIN {X 122.56, Y 50.93, Z 0.00, A 0, B 0, C 0} C_DIS
LIN {X 122.56, Y 51.26, Z 0.00, A 0, B 0, C 0} C_DIS
LIN {X 122.56, Y 51.58, Z 0.00, A 0, B 0, C 0} C_DIS
LIN {X 122.56, Y 51.91, Z 0.00, A 0, B 0, C 0} C_DIS
LIN {X 122.56, Y 52.24, Z 0.00, A 0, B 0, C 0} C_DIS
LIN {X 122.56, Y 52.57, Z 0.00, A 0, B 0, C 0} C_DIS
LIN {X 122.56, Y 52.89, Z 0.00, A 0, B 0, C 0} C_DIS
LIN {X 122.56, Y 53.22, Z 0.00, A 0, B 0, C 0} C_DIS
LIN {X 122.56, Y 53.55, Z 0.00, A 0, B 0, C 0} C_DIS
LIN {X 122.56, Y 53.88, Z 0.00, A 0, B 0, C 0} C_DIS
LIN {X 122.56, Y 54.21, Z 0.00, A 0, B 0, C 0} C_DIS
LIN {X 122.56, Y 54.53, Z 0.00, A 0, B 0, C 0} C_DIS
LIN {X 122.56, Y 54.86, Z 0.00, A 0, B 0, C 0} C_DIS
LIN {X 122.56, Y 55.19, Z 0.00, A 0, B 0, C 0} C_DIS
LIN {X 122.56, Y 55.52, Z 0.00, A 0, B 0, C 0} C_DIS
LIN {X 122.56, Y 55.84, Z 0.00, A 0, B 0, C 0} C_DIS
LIN {X 122.56, Y 56.17, Z 0.00, A 0, B 0, C 0} C_DIS
LIN {X 122.56, Y 56.50, Z 0.00, A 0, B 0, C 0} C_DIS
LIN {X 122.56, Y 56.83, Z 0.00, A 0, B 0, C 0} C_DIS
LIN {X 122.56, Y 57.15, Z 0.00, A 0, B 0, C 0} C_DIS
LIN {X 122.56, Y 57.48, Z 0.00, A 0, B 0, C 0} C_DIS
LIN {X 122.56, Y 57.81, Z 0.00, A 0, B 0, C 0} C_DIS
LIN {X 122.56, Y 58.14, Z 0.00, A 0, B 0, C 0} C_DIS
LIN {X 122.56, Y 58.46, Z 0.00, A 0, B 0, C 0} C_DIS
LIN {X 122.56, Y 58.79, Z 0.00, A 0, B 0, C 0} C_DIS
LIN {X 122.56, Y 59.12, Z 0.00, A 0, B 0, C 0} C_DIS
LIN {X 122.56, Y 59.45, Z 0.00, A 0, B 0, C 0} C_DIS
LIN {X 122.56, Y 59.78, Z 0.00, A 0, B 0, C 0} C_DIS
LIN {X 122.57, Y 60.11, Z 0.00, A 0, B 0, C 0} C_DIS
LIN {X 122.58, Y 60.44, Z 0.00, A 0, B 0, C 0} C_DIS
LIN {X 122.58, Y 60.77, Z 0.00, A 0, B 0, C 0} C_DIS
LIN {X 122.59, Y 61.10, Z 0.00, A 0, B 0, C 0} C_DIS
LIN {X 122.58, Y 61.42, Z 0.00, A 0, B 0, C 0} C_DIS
LIN {X 122.56, Y 61.75, Z 0.00, A 0, B 0, C 0} C_DIS
LIN {X 122.53, Y 62.07, Z 0.00, A 0, B 0, C 0} C_DIS
LIN {X 122.48, Y 62.39, Z 0.00, A 0, B 0, C 0} C_DIS
LIN {X 122.41, Y 62.70, Z 0.00, A 0, B 0, C 0} C_DIS
LIN {X 122.35, Y 63.02, Z 0.00, A 0, B 0, C 0} C_DIS
LIN {X 122.28, Y 63.33, Z 0.00, A 0, B 0, C 0} C_DIS
LIN {X 122.23, Y 63.65, Z 0.00, A 0, B 0, C 0} C_DIS
LIN {X 122.20, Y 63.97, Z 0.00, A 0, B 0, C 0} C_DIS
LIN {X 122.19, Y 64.30, Z 0.00, A 0, B 0, C 0} C_DIS
LIN {X 122.18, Y 64.63, Z 0.00, A 0, B 0, C 0} C_DIS
LIN {X 122.17, Y 64.96, Z 0.00, A 0, B 0, C 0} C_DIS
LIN {X 122.17, Y 65.29, Z 0.00, A 0, B 0, C 0} C_DIS
LIN {X 122.16, Y 65.62, Z 0.00, A 0, B 0, C 0} C_DIS
LIN {X 122.14, Y 65.94, Z 0.00, A 0, B 0, C 0} C_DIS
LIN {X 122.11, Y 66.26, Z 0.00, A 0, B 0, C 0} C_DIS
LIN {X 122.07, Y 66.58, Z 0.00, A 0, B 0, C 0} C_DIS
LIN {X 122.03, Y 66.90, Z 0.00, A 0, B 0, C 0} C_DIS
LIN {X 121.98, Y 67.22, Z 0.00, A 0, B 0, C 0} C_DIS
LIN {X 121.93, Y 67.53, Z 0.00, A 0, B 0, C 0} C_DIS
LIN {X 121.87, Y 67.85, Z 0.00, A 0, B 0, C 0} C_DIS
LIN {X 121.81, Y 68.16, Z 0.00, A 0, B 0, C 0} C_DIS
LIN {X 121.75, Y 68.47, Z 0.00, A 0, B 0, C 0} C_DIS
LIN {X 121.69, Y 68.78, Z 0.00, A 0, B 0, C 0} C_DIS
LIN {X 121.62, Y 69.10, Z 0.00, A 0, B 0, C 0} C_DIS
LIN {X 121.56, Y 69.41, Z 0.00, A 0, B 0, C 0} C_DIS
LIN {X 121.50, Y 69.72, Z 0.00, A 0, B 0, C 0} C_DIS
LIN {X 121.43, Y 70.04, Z 0.00, A 0, B 0, C 0} C_DIS
LIN {X 121.36, Y 70.35, Z 0.00, A 0, B 0, C 0} C_DIS
LIN {X 121.29, Y 70.66, Z 0.00, A 0, B 0, C 0} C_DIS
LIN {X 121.22, Y 70.97, Z 0.00, A 0, B 0, C 0} C_DIS
LIN {X 121.14, Y 71.27, Z 0.00, A 0, B 0, C 0} C_DIS
LIN {X 121.05, Y 71.57, Z 0.00, A 0, B 0, C 0} C_DIS
LIN {X 120.96, Y 71.86, Z 0.00, A 0, B 0, C 0} C_DIS
LIN {X 120.87, Y 72.15, Z 0.00, A 0, B 0, C 0} C_DIS
LIN {X 120.76, Y 72.44, Z 0.00, A 0, B 0, C 0} C_DIS
LIN {X 120.65, Y 72.72, Z 0.00, A 0, B 0, C 0} C_DIS
LIN {X 120.53, Y 72.99, Z 0.00, A 0, B 0, C 0} C_DIS
LIN {X 120.41, Y 73.27, Z 0.00, A 0, B 0, C 0} C_DIS
LIN {X 120.29, Y 73.54, Z 0.00, A 0, B 0, C 0} C_DIS
LIN {X 120.18, Y 73.81, Z 0.00, A 0, B 0, C 0} C_DIS
LIN {X 120.06, Y 74.09, Z 0.00, A 0, B 0, C 0} C_DIS
LIN {X 119.95, Y 74.37, Z 0.00, A 0, B 0, C 0} C_DIS
LIN {X 119.84, Y 74.65, Z 0.00, A 0, B 0, C 0} C_DIS
LIN {X 119.73, Y 74.94, Z 0.00, A 0, B 0, C 0} C_DIS
LIN {X 119.64, Y 75.23, Z 0.00, A 0, B 0, C 0} C_DIS
LIN {X 119.54, Y 75.52, Z 0.00, A 0, B 0, C 0} C_DIS
LIN {X 119.44, Y 75.81, Z 0.00, A 0, B 0, C 0} C_DIS
LIN {X 119.32, Y 76.09, Z 0.00, A 0, B 0, C 0} C_DIS
LIN {X 119.20, Y 76.35, Z 0.00, A 0, B 0, C 0} C_DIS
LIN {X 119.06, Y 76.60, Z 0.00, A 0, B 0, C 0} C_DIS
LIN {X 118.91, Y 76.84, Z 0.00, A 0, B 0, C 0} C_DIS
LIN {X 118.76, Y 77.08, Z 0.00, A 0, B 0, C 0} C_DIS
LIN {X 118.60, Y 77.31, Z 0.00, A 0, B 0, C 0} C_DIS
LIN {X 118.45, Y 77.54, Z 0.00, A 0, B 0, C 0} C_DIS
LIN {X 118.29, Y 77.78, Z 0.00, A 0, B 0, C 0} C_DIS
LIN {X 118.14, Y 78.01, Z 0.00, A 0, B 0, C 0} C_DIS
LIN {X 117.99, Y 78.24, Z 0.00, A 0, B 0, C 0} C_DIS
LIN {X 117.84, Y 78.48, Z 0.00, A 0, B 0, C 0} C_DIS
LIN {X 117.68, Y 78.71, Z 0.00, A 0, B 0, C 0} C_DIS
LIN {X 117.53, Y 78.94, Z 0.00, A 0, B 0, C 0} C_DIS
LIN {X 117.38, Y 79.17, Z 0.00, A 0, B 0, C 0} C_DIS
LIN {X 117.22, Y 79.40, Z 0.00, A 0, B 0, C 0} C_DIS
LIN {X 117.07, Y 79.63, Z 0.00, A 0, B 0, C 0} C_DIS
LIN {X 116.91, Y 79.86, Z 0.00, A 0, B 0, C 0} C_DIS
LIN {X 116.75, Y 80.08, Z 0.00, A 0, B 0, C 0} C_DIS
LIN {X 116.59, Y 80.30, Z 0.00, A 0, B 0, C 0} C_DIS
LIN {X 116.43, Y 80.51, Z 0.00, A 0, B 0, C 0} C_DIS
LIN {X 116.27, Y 80.73, Z 0.00, A 0, B 0, C 0} C_DIS
LIN {X 116.10, Y 80.94, Z 0.00, A 0, B 0, C 0} C_DIS
LIN {X 115.93, Y 81.14, Z 0.00, A 0, B 0, C 0} C_DIS
LIN {X 115.76, Y 81.34, Z 0.00, A 0, B 0, C 0} C_DIS
LIN {X 115.59, Y 81.54, Z 0.00, A 0, B 0, C 0} C_DIS
LIN {X 115.41, Y 81.73, Z 0.00, A 0, B 0, C 0} C_DIS
LIN {X 115.23, Y 81.92, Z 0.00, A 0, B 0, C 0} C_DIS
LIN {X 115.05, Y 82.10, Z 0.00, A 0, B 0, C 0} C_DIS
LIN {X 114.86, Y 82.28, Z 0.00, A 0, B 0, C 0} C_DIS
LIN {X 114.68, Y 82.45, Z 0.00, A 0, B 0, C 0} C_DIS
LIN {X 114.49, Y 82.62, Z 0.00, A 0, B 0, C 0} C_DIS
LIN {X 114.30, Y 82.78, Z 0.00, A 0, B 0, C 0} C_DIS
LIN {X 114.11, Y 82.93, Z 0.00, A 0, B 0, C 0} C_DIS
LIN {X 113.91, Y 83.08, Z 0.00, A 0, B 0, C 0} C_DIS
LIN {X 113.72, Y 83.22, Z 0.00, A 0, B 0, C 0} C_DIS
LIN {X 113.52, Y 83.36, Z 0.00, A 0, B 0, C 0} C_DIS
LIN {X 113.33, Y 83.49, Z 0.00, A 0, B 0, C 0} C_DIS
LIN {X 113.13, Y 83.62, Z 0.00, A 0, B 0, C 0} C_DIS
LIN {X 112.93, Y 83.74, Z 0.00, A 0, B 0, C 0} C_DIS
LIN {X 112.73, Y 83.86, Z 0.00, A 0, B 0, C 0} C_DIS
LIN {X 112.53, Y 83.98, Z 0.00, A 0, B 0, C 0} C_DIS
LIN {X 112.33, Y 84.09, Z 0.00, A 0, B 0, C 0} C_DIS
LIN {X 112.13, Y 84.21, Z 0.00, A 0, B 0, C 0} C_DIS
LIN {X 111.92, Y 84.32, Z 0.00, A 0, B 0, C 0} C_DIS
LIN {X 111.72, Y 84.43, Z 0.00, A 0, B 0, C 0} C_DIS
LIN {X 111.51, Y 84.54, Z 0.00, A 0, B 0, C 0} C_DIS
LIN {X 111.31, Y 84.65, Z 0.00, A 0, B 0, C 0} C_DIS
LIN {X 111.10, Y 84.75, Z 0.00, A 0, B 0, C 0} C_DIS
LIN {X 110.89, Y 84.85, Z 0.00, A 0, B 0, C 0} C_DIS
LIN {X 110.68, Y 84.94, Z 0.00, A 0, B 0, C 0} C_DIS
LIN {X 110.47, Y 85.02, Z 0.00, A 0, B 0, C 0} C_DIS
LIN {X 110.26, Y 85.10, Z 0.00, A 0, B 0, C 0} C_DIS
LIN {X 110.05, Y 85.17, Z 0.00, A 0, B 0, C 0} C_DIS
LIN {X 109.84, Y 85.23, Z 0.00, A 0, B 0, C 0} C_DIS
LIN {X 109.62, Y 85.29, Z 0.00, A 0, B 0, C 0} C_DIS
LIN {X 109.41, Y 85.34, Z 0.00, A 0, B 0, C 0} C_DIS
LIN {X 109.20, Y 85.40, Z 0.00, A 0, B 0, C 0} C_DIS
LIN {X 108.98, Y 85.46, Z 0.00, A 0, B 0, C 0} C_DIS
LIN {X 108.77, Y 85.53, Z 0.00, A 0, B 0, C 0} C_DIS
LIN {X 108.56, Y 85.61, Z 0.00, A 0, B 0, C 0} C_DIS
LIN {X 108.36, Y 85.70, Z 0.00, A 0, B 0, C 0} C_DIS
LIN {X 108.15, Y 85.82, Z 0.00, A 0, B 0, C 0} C_DIS
LIN {X 108.15, Y 85.82, Z 10.00, A 0, B 0, C 0}

; ----- Contour 3 -----
PTP {X 157.17, Y 257.39, Z 10.00, A 0, B 0, C 0}
LIN {X 157.17, Y 257.39, Z 0.00, A 0, B 0, C 0}
LIN {X 157.35, Y 257.22, Z 0.00, A 0, B 0, C 0} C_DIS
LIN {X 157.51, Y 257.01, Z 0.00, A 0, B 0, C 0} C_DIS
LIN {X 157.66, Y 256.77, Z 0.00, A 0, B 0, C 0} C_DIS
LIN {X 157.82, Y 256.54, Z 0.00, A 0, B 0, C 0} C_DIS
LIN {X 157.96, Y 256.29, Z 0.00, A 0, B 0, C 0} C_DIS
LIN {X 158.03, Y 255.99, Z 0.00, A 0, B 0, C 0} C_DIS
LIN {X 158.04, Y 255.65, Z 0.00, A 0, B 0, C 0} C_DIS
LIN {X 158.04, Y 255.32, Z 0.00, A 0, B 0, C 0} C_DIS
LIN {X 158.01, Y 255.00, Z 0.00, A 0, B 0, C 0} C_DIS
LIN {X 157.94, Y 254.70, Z 0.00, A 0, B 0, C 0} C_DIS
LIN {X 157.83, Y 254.41, Z 0.00, A 0, B 0, C 0} C_DIS
LIN {X 157.71, Y 254.14, Z 0.00, A 0, B 0, C 0} C_DIS
LIN {X 157.58, Y 253.87, Z 0.00, A 0, B 0, C 0} C_DIS
LIN {X 157.45, Y 253.61, Z 0.00, A 0, B 0, C 0} C_DIS
LIN {X 157.31, Y 253.36, Z 0.00, A 0, B 0, C 0} C_DIS
LIN {X 157.17, Y 253.12, Z 0.00, A 0, B 0, C 0} C_DIS
LIN {X 157.01, Y 252.89, Z 0.00, A 0, B 0, C 0} C_DIS
LIN {X 156.85, Y 252.67, Z 0.00, A 0, B 0, C 0} C_DIS
LIN {X 156.68, Y 252.46, Z 0.00, A 0, B 0, C 0} C_DIS
LIN {X 156.51, Y 252.27, Z 0.00, A 0, B 0, C 0} C_DIS
LIN {X 156.33, Y 252.08, Z 0.00, A 0, B 0, C 0} C_DIS
LIN {X 156.14, Y 251.91, Z 0.00, A 0, B 0, C 0} C_DIS
LIN {X 155.96, Y 251.73, Z 0.00, A 0, B 0, C 0} C_DIS
LIN {X 155.78, Y 251.55, Z 0.00, A 0, B 0, C 0} C_DIS
LIN {X 155.60, Y 251.37, Z 0.00, A 0, B 0, C 0} C_DIS
LIN {X 155.42, Y 251.18, Z 0.00, A 0, B 0, C 0} C_DIS
LIN {X 155.24, Y 250.99, Z 0.00, A 0, B 0, C 0} C_DIS
LIN {X 155.06, Y 250.81, Z 0.00, A 0, B 0, C 0} C_DIS
LIN {X 154.88, Y 250.63, Z 0.00, A 0, B 0, C 0} C_DIS
LIN {X 154.69, Y 250.47, Z 0.00, A 0, B 0, C 0} C_DIS
LIN {X 154.50, Y 250.32, Z 0.00, A 0, B 0, C 0} C_DIS
LIN {X 154.30, Y 250.19, Z 0.00, A 0, B 0, C 0} C_DIS
LIN {X 154.10, Y 250.06, Z 0.00, A 0, B 0, C 0} C_DIS
LIN {X 153.91, Y 249.89, Z 0.00, A 0, B 0, C 0} C_DIS
LIN {X 153.73, Y 249.72, Z 0.00, A 0, B 0, C 0} C_DIS
LIN {X 153.53, Y 249.59, Z 0.00, A 0, B 0, C 0} C_DIS
LIN {X 153.32, Y 249.50, Z 0.00, A 0, B 0, C 0} C_DIS
LIN {X 153.11, Y 249.42, Z 0.00, A 0, B 0, C 0} C_DIS
LIN {X 152.91, Y 249.30, Z 0.00, A 0, B 0, C 0} C_DIS
LIN {X 152.71, Y 249.16, Z 0.00, A 0, B 0, C 0} C_DIS
LIN {X 152.51, Y 249.04, Z 0.00, A 0, B 0, C 0} C_DIS
LIN {X 152.30, Y 248.95, Z 0.00, A 0, B 0, C 0} C_DIS
LIN {X 152.09, Y 248.88, Z 0.00, A 0, B 0, C 0} C_DIS
LIN {X 151.88, Y 248.80, Z 0.00, A 0, B 0, C 0} C_DIS
LIN {X 151.67, Y 248.69, Z 0.00, A 0, B 0, C 0} C_DIS
LIN {X 151.47, Y 248.55, Z 0.00, A 0, B 0, C 0} C_DIS
LIN {X 151.27, Y 248.43, Z 0.00, A 0, B 0, C 0} C_DIS
LIN {X 151.07, Y 248.32, Z 0.00, A 0, B 0, C 0} C_DIS
LIN {X 150.86, Y 248.24, Z 0.00, A 0, B 0, C 0} C_DIS
LIN {X 150.64, Y 248.16, Z 0.00, A 0, B 0, C 0} C_DIS
LIN {X 150.43, Y 248.09, Z 0.00, A 0, B 0, C 0} C_DIS
LIN {X 150.22, Y 248.02, Z 0.00, A 0, B 0, C 0} C_DIS
LIN {X 150.01, Y 247.96, Z 0.00, A 0, B 0, C 0} C_DIS
LIN {X 149.79, Y 247.91, Z 0.00, A 0, B 0, C 0} C_DIS
LIN {X 149.58, Y 247.88, Z 0.00, A 0, B 0, C 0} C_DIS
LIN {X 149.36, Y 247.84, Z 0.00, A 0, B 0, C 0} C_DIS
LIN {X 149.15, Y 247.78, Z 0.00, A 0, B 0, C 0} C_DIS
LIN {X 148.94, Y 247.71, Z 0.00, A 0, B 0, C 0} C_DIS
LIN {X 148.73, Y 247.62, Z 0.00, A 0, B 0, C 0} C_DIS
LIN {X 148.52, Y 247.52, Z 0.00, A 0, B 0, C 0} C_DIS
LIN {X 148.31, Y 247.43, Z 0.00, A 0, B 0, C 0} C_DIS
LIN {X 148.09, Y 247.36, Z 0.00, A 0, B 0, C 0} C_DIS
LIN {X 147.88, Y 247.31, Z 0.00, A 0, B 0, C 0} C_DIS
LIN {X 147.66, Y 247.29, Z 0.00, A 0, B 0, C 0} C_DIS
LIN {X 147.45, Y 247.28, Z 0.00, A 0, B 0, C 0} C_DIS
LIN {X 147.23, Y 247.26, Z 0.00, A 0, B 0, C 0} C_DIS
LIN {X 147.01, Y 247.24, Z 0.00, A 0, B 0, C 0} C_DIS
LIN {X 146.80, Y 247.19, Z 0.00, A 0, B 0, C 0} C_DIS
LIN {X 146.59, Y 247.14, Z 0.00, A 0, B 0, C 0} C_DIS
LIN {X 146.37, Y 247.07, Z 0.00, A 0, B 0, C 0} C_DIS
LIN {X 146.16, Y 246.98, Z 0.00, A 0, B 0, C 0} C_DIS
LIN {X 145.95, Y 246.89, Z 0.00, A 0, B 0, C 0} C_DIS
LIN {X 145.74, Y 246.80, Z 0.00, A 0, B 0, C 0} C_DIS
LIN {X 145.53, Y 246.72, Z 0.00, A 0, B 0, C 0} C_DIS
LIN {X 145.32, Y 246.66, Z 0.00, A 0, B 0, C 0} C_DIS
LIN {X 145.10, Y 246.63, Z 0.00, A 0, B 0, C 0} C_DIS
LIN {X 144.89, Y 246.61, Z 0.00, A 0, B 0, C 0} C_DIS
LIN {X 144.67, Y 246.60, Z 0.00, A 0, B 0, C 0} C_DIS
LIN {X 144.45, Y 246.61, Z 0.00, A 0, B 0, C 0} C_DIS
LIN {X 144.23, Y 246.62, Z 0.00, A 0, B 0, C 0} C_DIS
LIN {X 144.01, Y 246.62, Z 0.00, A 0, B 0, C 0} C_DIS
LIN {X 143.80, Y 246.61, Z 0.00, A 0, B 0, C 0} C_DIS
LIN {X 143.58, Y 246.59, Z 0.00, A 0, B 0, C 0} C_DIS
LIN {X 143.37, Y 246.55, Z 0.00, A 0, B 0, C 0} C_DIS
LIN {X 143.15, Y 246.50, Z 0.00, A 0, B 0, C 0} C_DIS
LIN {X 142.94, Y 246.43, Z 0.00, A 0, B 0, C 0} C_DIS
LIN {X 142.73, Y 246.35, Z 0.00, A 0, B 0, C 0} C_DIS
LIN {X 142.52, Y 246.26, Z 0.00, A 0, B 0, C 0} C_DIS
LIN {X 142.31, Y 246.16, Z 0.00, A 0, B 0, C 0} C_DIS
LIN {X 142.10, Y 246.08, Z 0.00, A 0, B 0, C 0} C_DIS
LIN {X 141.89, Y 246.02, Z 0.00, A 0, B 0, C 0} C_DIS
LIN {X 141.67, Y 245.99, Z 0.00, A 0, B 0, C 0} C_DIS
LIN {X 141.45, Y 245.97, Z 0.00, A 0, B 0, C 0} C_DIS
LIN {X 141.24, Y 245.93, Z 0.00, A 0, B 0, C 0} C_DIS
LIN {X 141.03, Y 245.84, Z 0.00, A 0, B 0, C 0} C_DIS
LIN {X 140.83, Y 245.68, Z 0.00, A 0, B 0, C 0} C_DIS
LIN {X 140.67, Y 245.47, Z 0.00, A 0, B 0, C 0} C_DIS
LIN {X 140.56, Y 245.20, Z 0.00, A 0, B 0, C 0} C_DIS
LIN {X 140.51, Y 244.89, Z 0.00, A 0, B 0, C 0} C_DIS
LIN {X 140.49, Y 244.55, Z 0.00, A 0, B 0, C 0} C_DIS
LIN {X 140.48, Y 244.21, Z 0.00, A 0, B 0, C 0} C_DIS
LIN {X 140.48, Y 243.88, Z 0.00, A 0, B 0, C 0} C_DIS
LIN {X 140.49, Y 243.56, Z 0.00, A 0, B 0, C 0} C_DIS
LIN {X 140.51, Y 243.24, Z 0.00, A 0, B 0, C 0} C_DIS
LIN {X 140.55, Y 242.92, Z 0.00, A 0, B 0, C 0} C_DIS
LIN {X 140.60, Y 242.60, Z 0.00, A 0, B 0, C 0} C_DIS
LIN {X 140.66, Y 242.28, Z 0.00, A 0, B 0, C 0} C_DIS
LIN {X 140.72, Y 241.97, Z 0.00, A 0, B 0, C 0} C_DIS
LIN {X 140.78, Y 241.65, Z 0.00, A 0, B 0, C 0} C_DIS
LIN {X 140.83, Y 241.33, Z 0.00, A 0, B 0, C 0} C_DIS
LIN {X 140.87, Y 241.01, Z 0.00, A 0, B 0, C 0} C_DIS
LIN {X 140.90, Y 240.68, Z 0.00, A 0, B 0, C 0} C_DIS
LIN {X 140.91, Y 240.36, Z 0.00, A 0, B 0, C 0} C_DIS
LIN {X 140.92, Y 240.03, Z 0.00, A 0, B 0, C 0} C_DIS
LIN {X 140.92, Y 239.70, Z 0.00, A 0, B 0, C 0} C_DIS
LIN {X 140.91, Y 239.37, Z 0.00, A 0, B 0, C 0} C_DIS
LIN {X 140.91, Y 239.04, Z 0.00, A 0, B 0, C 0} C_DIS
LIN {X 140.91, Y 238.72, Z 0.00, A 0, B 0, C 0} C_DIS
LIN {X 140.92, Y 238.39, Z 0.00, A 0, B 0, C 0} C_DIS
LIN {X 140.94, Y 238.07, Z 0.00, A 0, B 0, C 0} C_DIS
LIN {X 140.98, Y 237.74, Z 0.00, A 0, B 0, C 0} C_DIS
LIN {X 141.02, Y 237.43, Z 0.00, A 0, B 0, C 0} C_DIS
LIN {X 141.08, Y 237.11, Z 0.00, A 0, B 0, C 0} C_DIS
LIN {X 141.14, Y 236.79, Z 0.00, A 0, B 0, C 0} C_DIS
LIN {X 141.20, Y 236.47, Z 0.00, A 0, B 0, C 0} C_DIS
LIN {X 141.25, Y 236.15, Z 0.00, A 0, B 0, C 0} C_DIS
LIN {X 141.30, Y 235.83, Z 0.00, A 0, B 0, C 0} C_DIS
LIN {X 141.33, Y 235.51, Z 0.00, A 0, B 0, C 0} C_DIS
LIN {X 141.34, Y 235.19, Z 0.00, A 0, B 0, C 0} C_DIS
LIN {X 141.35, Y 234.86, Z 0.00, A 0, B 0, C 0} C_DIS
LIN {X 141.35, Y 234.53, Z 0.00, A 0, B 0, C 0} C_DIS
LIN {X 141.35, Y 234.20, Z 0.00, A 0, B 0, C 0} C_DIS
LIN {X 141.34, Y 233.87, Z 0.00, A 0, B 0, C 0} C_DIS
LIN {X 141.35, Y 233.55, Z 0.00, A 0, B 0, C 0} C_DIS
LIN {X 141.35, Y 233.22, Z 0.00, A 0, B 0, C 0} C_DIS
LIN {X 141.37, Y 232.89, Z 0.00, A 0, B 0, C 0} C_DIS
LIN {X 141.40, Y 232.57, Z 0.00, A 0, B 0, C 0} C_DIS
LIN {X 141.45, Y 232.25, Z 0.00, A 0, B 0, C 0} C_DIS
LIN {X 141.50, Y 231.93, Z 0.00, A 0, B 0, C 0} C_DIS
LIN {X 141.56, Y 231.62, Z 0.00, A 0, B 0, C 0} C_DIS
LIN {X 141.62, Y 231.30, Z 0.00, A 0, B 0, C 0} C_DIS
LIN {X 141.68, Y 230.98, Z 0.00, A 0, B 0, C 0} C_DIS
LIN {X 141.72, Y 230.66, Z 0.00, A 0, B 0, C 0} C_DIS
LIN {X 141.75, Y 230.34, Z 0.00, A 0, B 0, C 0} C_DIS
LIN {X 141.77, Y 230.01, Z 0.00, A 0, B 0, C 0} C_DIS
LIN {X 141.78, Y 229.69, Z 0.00, A 0, B 0, C 0} C_DIS
LIN {X 141.79, Y 229.36, Z 0.00, A 0, B 0, C 0} C_DIS
LIN {X 141.78, Y 229.03, Z 0.00, A 0, B 0, C 0} C_DIS
LIN {X 141.78, Y 228.70, Z 0.00, A 0, B 0, C 0} C_DIS
LIN {X 141.78, Y 228.37, Z 0.00, A 0, B 0, C 0} C_DIS
LIN {X 141.79, Y 228.05, Z 0.00, A 0, B 0, C 0} C_DIS
LIN {X 141.80, Y 227.72, Z 0.00, A 0, B 0, C 0} C_DIS
LIN {X 141.83, Y 227.40, Z 0.00, A 0, B 0, C 0} C_DIS
LIN {X 141.87, Y 227.08, Z 0.00, A 0, B 0, C 0} C_DIS
LIN {X 141.92, Y 226.76, Z 0.00, A 0, B 0, C 0} C_DIS
LIN {X 141.98, Y 226.44, Z 0.00, A 0, B 0, C 0} C_DIS
LIN {X 142.04, Y 226.12, Z 0.00, A 0, B 0, C 0} C_DIS
LIN {X 142.09, Y 225.81, Z 0.00, A 0, B 0, C 0} C_DIS
LIN {X 142.14, Y 225.49, Z 0.00, A 0, B 0, C 0} C_DIS
LIN {X 142.18, Y 225.17, Z 0.00, A 0, B 0, C 0} C_DIS
LIN {X 142.21, Y 224.84, Z 0.00, A 0, B 0, C 0} C_DIS
LIN {X 142.22, Y 224.52, Z 0.00, A 0, B 0, C 0} C_DIS
LIN {X 142.23, Y 224.19, Z 0.00, A 0, B 0, C 0} C_DIS
LIN {X 142.23, Y 223.86, Z 0.00, A 0, B 0, C 0} C_DIS
LIN {X 142.22, Y 223.53, Z 0.00, A 0, B 0, C 0} C_DIS
LIN {X 142.21, Y 223.20, Z 0.00, A 0, B 0, C 0} C_DIS
LIN {X 142.21, Y 222.88, Z 0.00, A 0, B 0, C 0} C_DIS
LIN {X 142.23, Y 222.55, Z 0.00, A 0, B 0, C 0} C_DIS
LIN {X 142.26, Y 222.23, Z 0.00, A 0, B 0, C 0} C_DIS
LIN {X 142.30, Y 221.90, Z 0.00, A 0, B 0, C 0} C_DIS
LIN {X 142.35, Y 221.58, Z 0.00, A 0, B 0, C 0} C_DIS
LIN {X 142.40, Y 221.27, Z 0.00, A 0, B 0, C 0} C_DIS
LIN {X 142.46, Y 220.95, Z 0.00, A 0, B 0, C 0} C_DIS
LIN {X 142.52, Y 220.63, Z 0.00, A 0, B 0, C 0} C_DIS
LIN {X 142.57, Y 220.32, Z 0.00, A 0, B 0, C 0} C_DIS
LIN {X 142.61, Y 219.99, Z 0.00, A 0, B 0, C 0} C_DIS
LIN {X 142.64, Y 219.67, Z 0.00, A 0, B 0, C 0} C_DIS
LIN {X 142.66, Y 219.35, Z 0.00, A 0, B 0, C 0} C_DIS
LIN {X 142.66, Y 219.02, Z 0.00, A 0, B 0, C 0} C_DIS
LIN {X 142.66, Y 218.69, Z 0.00, A 0, B 0, C 0} C_DIS
LIN {X 142.65, Y 218.36, Z 0.00, A 0, B 0, C 0} C_DIS
LIN {X 142.65, Y 218.03, Z 0.00, A 0, B 0, C 0} C_DIS
LIN {X 142.65, Y 217.70, Z 0.00, A 0, B 0, C 0} C_DIS
LIN {X 142.66, Y 217.38, Z 0.00, A 0, B 0, C 0} C_DIS
LIN {X 142.69, Y 217.05, Z 0.00, A 0, B 0, C 0} C_DIS
LIN {X 142.72, Y 216.73, Z 0.00, A 0, B 0, C 0} C_DIS
LIN {X 142.77, Y 216.41, Z 0.00, A 0, B 0, C 0} C_DIS
LIN {X 142.82, Y 216.09, Z 0.00, A 0, B 0, C 0} C_DIS
LIN {X 142.88, Y 215.78, Z 0.00, A 0, B 0, C 0} C_DIS
LIN {X 142.94, Y 215.46, Z 0.00, A 0, B 0, C 0} C_DIS
LIN {X 142.99, Y 215.14, Z 0.00, A 0, B 0, C 0} C_DIS
LIN {X 143.04, Y 214.82, Z 0.00, A 0, B 0, C 0} C_DIS
LIN {X 143.07, Y 214.50, Z 0.00, A 0, B 0, C 0} C_DIS
LIN {X 143.09, Y 214.17, Z 0.00, A 0, B 0, C 0} C_DIS
LIN {X 143.10, Y 213.85, Z 0.00, A 0, B 0, C 0} C_DIS
LIN {X 143.10, Y 213.52, Z 0.00, A 0, B 0, C 0} C_DIS
LIN {X 143.09, Y 213.19, Z 0.00, A 0, B 0, C 0} C_DIS
LIN {X 143.08, Y 212.86, Z 0.00, A 0, B 0, C 0} C_DIS
LIN {X 143.09, Y 212.53, Z 0.00, A 0, B 0, C 0} C_DIS
LIN {X 143.09, Y 212.21, Z 0.00, A 0, B 0, C 0} C_DIS
LIN {X 143.11, Y 211.88, Z 0.00, A 0, B 0, C 0} C_DIS
LIN {X 143.15, Y 211.56, Z 0.00, A 0, B 0, C 0} C_DIS
LIN {X 143.19, Y 211.24, Z 0.00, A 0, B 0, C 0} C_DIS
LIN {X 143.25, Y 210.92, Z 0.00, A 0, B 0, C 0} C_DIS
LIN {X 143.31, Y 210.60, Z 0.00, A 0, B 0, C 0} C_DIS
LIN {X 143.36, Y 210.29, Z 0.00, A 0, B 0, C 0} C_DIS
LIN {X 143.42, Y 209.97, Z 0.00, A 0, B 0, C 0} C_DIS
LIN {X 143.46, Y 209.65, Z 0.00, A 0, B 0, C 0} C_DIS
LIN {X 143.50, Y 209.33, Z 0.00, A 0, B 0, C 0} C_DIS
LIN {X 143.52, Y 209.00, Z 0.00, A 0, B 0, C 0} C_DIS
LIN {X 143.53, Y 208.68, Z 0.00, A 0, B 0, C 0} C_DIS
LIN {X 143.53, Y 208.35, Z 0.00, A 0, B 0, C 0} C_DIS
LIN {X 143.52, Y 208.02, Z 0.00, A 0, B 0, C 0} C_DIS
LIN {X 143.52, Y 207.69, Z 0.00, A 0, B 0, C 0} C_DIS
LIN {X 143.52, Y 207.36, Z 0.00, A 0, B 0, C 0} C_DIS
LIN {X 143.53, Y 207.03, Z 0.00, A 0, B 0, C 0} C_DIS
LIN {X 143.55, Y 206.71, Z 0.00, A 0, B 0, C 0} C_DIS
LIN {X 143.58, Y 206.39, Z 0.00, A 0, B 0, C 0} C_DIS
LIN {X 143.62, Y 206.06, Z 0.00, A 0, B 0, C 0} C_DIS
LIN {X 143.66, Y 205.74, Z 0.00, A 0, B 0, C 0} C_DIS
LIN {X 143.73, Y 205.43, Z 0.00, A 0, B 0, C 0} C_DIS
LIN {X 143.80, Y 205.12, Z 0.00, A 0, B 0, C 0} C_DIS
LIN {X 143.92, Y 204.85, Z 0.00, A 0, B 0, C 0} C_DIS
LIN {X 144.07, Y 204.62, Z 0.00, A 0, B 0, C 0} C_DIS
LIN {X 144.22, Y 204.38, Z 0.00, A 0, B 0, C 0} C_DIS
LIN {X 144.38, Y 204.16, Z 0.00, A 0, B 0, C 0} C_DIS
LIN {X 144.55, Y 203.95, Z 0.00, A 0, B 0, C 0} C_DIS
LIN {X 144.72, Y 203.76, Z 0.00, A 0, B 0, C 0} C_DIS
LIN {X 144.90, Y 203.57, Z 0.00, A 0, B 0, C 0} C_DIS
LIN {X 145.08, Y 203.38, Z 0.00, A 0, B 0, C 0} C_DIS
LIN {X 145.26, Y 203.20, Z 0.00, A 0, B 0, C 0} C_DIS
LIN {X 145.44, Y 203.02, Z 0.00, A 0, B 0, C 0} C_DIS
LIN {X 145.63, Y 202.84, Z 0.00, A 0, B 0, C 0} C_DIS
LIN {X 145.81, Y 202.66, Z 0.00, A 0, B 0, C 0} C_DIS
LIN {X 145.99, Y 202.48, Z 0.00, A 0, B 0, C 0} C_DIS
LIN {X 146.17, Y 202.30, Z 0.00, A 0, B 0, C 0} C_DIS
LIN {X 146.35, Y 202.12, Z 0.00, A 0, B 0, C 0} C_DIS
LIN {X 146.53, Y 201.94, Z 0.00, A 0, B 0, C 0} C_DIS
LIN {X 146.71, Y 201.76, Z 0.00, A 0, B 0, C 0} C_DIS
LIN {X 146.89, Y 201.57, Z 0.00, A 0, B 0, C 0} C_DIS
LIN {X 147.07, Y 201.39, Z 0.00, A 0, B 0, C 0} C_DIS
LIN {X 147.26, Y 201.21, Z 0.00, A 0, B 0, C 0} C_DIS
LIN {X 147.44, Y 201.03, Z 0.00, A 0, B 0, C 0} C_DIS
LIN {X 147.62, Y 200.84, Z 0.00, A 0, B 0, C 0} C_DIS
LIN {X 147.80, Y 200.66, Z 0.00, A 0, B 0, C 0} C_DIS
LIN {X 147.98, Y 200.48, Z 0.00, A 0, B 0, C 0} C_DIS
LIN {X 148.16, Y 200.30, Z 0.00, A 0, B 0, C 0} C_DIS
LIN {X 148.34, Y 200.12, Z 0.00, A 0, B 0, C 0} C_DIS
LIN {X 148.52, Y 199.94, Z 0.00, A 0, B 0, C 0} C_DIS
LIN {X 148.71, Y 199.76, Z 0.00, A 0, B 0, C 0} C_DIS
LIN {X 148.89, Y 199.58, Z 0.00, A 0, B 0, C 0} C_DIS
LIN {X 149.04, Y 199.36, Z 0.00, A 0, B 0, C 0} C_DIS
LIN {X 149.20, Y 199.12, Z 0.00, A 0, B 0, C 0} C_DIS
LIN {X 149.36, Y 198.90, Z 0.00, A 0, B 0, C 0} C_DIS
LIN {X 149.53, Y 198.70, Z 0.00, A 0, B 0, C 0} C_DIS
LIN {X 149.71, Y 198.52, Z 0.00, A 0, B 0, C 0} C_DIS
LIN {X 149.89, Y 198.34, Z 0.00, A 0, B 0, C 0} C_DIS
LIN {X 150.08, Y 198.17, Z 0.00, A 0, B 0, C 0} C_DIS
LIN {X 150.26, Y 197.99, Z 0.00, A 0, B 0, C 0} C_DIS
LIN {X 150.44, Y 197.80, Z 0.00, A 0, B 0, C 0} C_DIS
LIN {X 150.61, Y 197.60, Z 0.00, A 0, B 0, C 0} C_DIS
LIN {X 150.78, Y 197.39, Z 0.00, A 0, B 0, C 0} C_DIS
LIN {X 150.94, Y 197.18, Z 0.00, A 0, B 0, C 0} C_DIS
LIN {X 151.09, Y 196.95, Z 0.00, A 0, B 0, C 0} C_DIS
LIN {X 151.24, Y 196.71, Z 0.00, A 0, B 0, C 0} C_DIS
LIN {X 151.39, Y 196.47, Z 0.00, A 0, B 0, C 0} C_DIS
LIN {X 151.55, Y 196.24, Z 0.00, A 0, B 0, C 0} C_DIS
LIN {X 151.70, Y 196.00, Z 0.00, A 0, B 0, C 0} C_DIS
LIN {X 151.85, Y 195.77, Z 0.00, A 0, B 0, C 0} C_DIS
LIN {X 152.01, Y 195.54, Z 0.00, A 0, B 0, C 0} C_DIS
LIN {X 152.16, Y 195.31, Z 0.00, A 0, B 0, C 0} C_DIS
LIN {X 152.32, Y 195.09, Z 0.00, A 0, B 0, C 0} C_DIS
LIN {X 152.49, Y 194.88, Z 0.00, A 0, B 0, C 0} C_DIS
LIN {X 152.66, Y 194.68, Z 0.00, A 0, B 0, C 0} C_DIS
LIN {X 152.83, Y 194.49, Z 0.00, A 0, B 0, C 0} C_DIS
LIN {X 153.02, Y 194.31, Z 0.00, A 0, B 0, C 0} C_DIS
LIN {X 153.20, Y 194.14, Z 0.00, A 0, B 0, C 0} C_DIS
LIN {X 153.39, Y 193.97, Z 0.00, A 0, B 0, C 0} C_DIS
LIN {X 153.57, Y 193.79, Z 0.00, A 0, B 0, C 0} C_DIS
LIN {X 153.74, Y 193.58, Z 0.00, A 0, B 0, C 0} C_DIS
LIN {X 153.89, Y 193.35, Z 0.00, A 0, B 0, C 0} C_DIS
LIN {X 154.03, Y 193.10, Z 0.00, A 0, B 0, C 0} C_DIS
LIN {X 154.16, Y 192.83, Z 0.00, A 0, B 0, C 0} C_DIS
LIN {X 154.27, Y 192.56, Z 0.00, A 0, B 0, C 0} C_DIS
LIN {X 154.39, Y 192.28, Z 0.00, A 0, B 0, C 0} C_DIS
LIN {X 154.50, Y 192.00, Z 0.00, A 0, B 0, C 0} C_DIS
LIN {X 154.62, Y 191.72, Z 0.00, A 0, B 0, C 0} C_DIS
LIN {X 154.76, Y 191.47, Z 0.00, A 0, B 0, C 0} C_DIS
LIN {X 154.90, Y 191.22, Z 0.00, A 0, B 0, C 0} C_DIS
LIN {X 155.04, Y 190.98, Z 0.00, A 0, B 0, C 0} C_DIS
LIN {X 155.19, Y 190.74, Z 0.00, A 0, B 0, C 0} C_DIS
LIN {X 155.34, Y 190.51, Z 0.00, A 0, B 0, C 0} C_DIS
LIN {X 155.50, Y 190.27, Z 0.00, A 0, B 0, C 0} C_DIS
LIN {X 155.65, Y 190.05, Z 0.00, A 0, B 0, C 0} C_DIS
LIN {X 155.81, Y 189.82, Z 0.00, A 0, B 0, C 0} C_DIS
LIN {X 155.97, Y 189.59, Z 0.00, A 0, B 0, C 0} C_DIS
LIN {X 156.12, Y 189.36, Z 0.00, A 0, B 0, C 0} C_DIS
LIN {X 156.28, Y 189.13, Z 0.00, A 0, B 0, C 0} C_DIS
LIN {X 156.42, Y 188.89, Z 0.00, A 0, B 0, C 0} C_DIS
LIN {X 156.57, Y 188.64, Z 0.00, A 0, B 0, C 0} C_DIS
LIN {X 156.70, Y 188.38, Z 0.00, A 0, B 0, C 0} C_DIS
LIN {X 156.82, Y 188.11, Z 0.00, A 0, B 0, C 0} C_DIS
LIN {X 156.94, Y 187.84, Z 0.00, A 0, B 0, C 0} C_DIS
LIN {X 157.05, Y 187.56, Z 0.00, A 0, B 0, C 0} C_DIS
LIN {X 157.17, Y 187.28, Z 0.00, A 0, B 0, C 0} C_DIS
LIN {X 157.29, Y 187.01, Z 0.00, A 0, B 0, C 0} C_DIS
LIN {X 157.43, Y 186.76, Z 0.00, A 0, B 0, C 0} C_DIS
LIN {X 157.57, Y 186.51, Z 0.00, A 0, B 0, C 0} C_DIS
LIN {X 157.72, Y 186.27, Z 0.00, A 0, B 0, C 0} C_DIS
LIN {X 157.86, Y 186.03, Z 0.00, A 0, B 0, C 0} C_DIS
LIN {X 158.00, Y 185.78, Z 0.00, A 0, B 0, C 0} C_DIS
LIN {X 158.12, Y 185.51, Z 0.00, A 0, B 0, C 0} C_DIS
LIN {X 158.24, Y 185.22, Z 0.00, A 0, B 0, C 0} C_DIS
LIN {X 158.35, Y 184.94, Z 0.00, A 0, B 0, C 0} C_DIS
LIN {X 158.45, Y 184.66, Z 0.00, A 0, B 0, C 0} C_DIS
LIN {X 158.54, Y 184.36, Z 0.00, A 0, B 0, C 0} C_DIS
LIN {X 158.62, Y 184.05, Z 0.00, A 0, B 0, C 0} C_DIS
LIN {X 158.73, Y 183.77, Z 0.00, A 0, B 0, C 0} C_DIS
LIN {X 158.85, Y 183.49, Z 0.00, A 0, B 0, C 0} C_DIS
LIN {X 158.93, Y 183.19, Z 0.00, A 0, B 0, C 0} C_DIS
LIN {X 159.01, Y 182.89, Z 0.00, A 0, B 0, C 0} C_DIS
LIN {X 159.11, Y 182.60, Z 0.00, A 0, B 0, C 0} C_DIS
LIN {X 159.23, Y 182.32, Z 0.00, A 0, B 0, C 0} C_DIS
LIN {X 159.33, Y 182.03, Z 0.00, A 0, B 0, C 0} C_DIS
LIN {X 159.41, Y 181.73, Z 0.00, A 0, B 0, C 0} C_DIS
LIN {X 159.49, Y 181.42, Z 0.00, A 0, B 0, C 0} C_DIS
LIN {X 159.61, Y 181.15, Z 0.00, A 0, B 0, C 0} C_DIS
LIN {X 159.72, Y 180.87, Z 0.00, A 0, B 0, C 0} C_DIS
LIN {X 159.80, Y 180.56, Z 0.00, A 0, B 0, C 0} C_DIS
LIN {X 159.88, Y 180.26, Z 0.00, A 0, B 0, C 0} C_DIS
LIN {X 159.98, Y 179.97, Z 0.00, A 0, B 0, C 0} C_DIS
LIN {X 160.10, Y 179.69, Z 0.00, A 0, B 0, C 0} C_DIS
LIN {X 160.20, Y 179.40, Z 0.00, A 0, B 0, C 0} C_DIS
LIN {X 160.27, Y 179.10, Z 0.00, A 0, B 0, C 0} C_DIS
LIN {X 160.33, Y 178.78, Z 0.00, A 0, B 0, C 0} C_DIS
LIN {X 160.40, Y 178.47, Z 0.00, A 0, B 0, C 0} C_DIS
LIN {X 160.48, Y 178.16, Z 0.00, A 0, B 0, C 0} C_DIS
LIN {X 160.57, Y 177.87, Z 0.00, A 0, B 0, C 0} C_DIS
LIN {X 160.64, Y 177.56, Z 0.00, A 0, B 0, C 0} C_DIS
LIN {X 160.69, Y 177.24, Z 0.00, A 0, B 0, C 0} C_DIS
LIN {X 160.76, Y 176.93, Z 0.00, A 0, B 0, C 0} C_DIS
LIN {X 160.87, Y 176.64, Z 0.00, A 0, B 0, C 0} C_DIS
LIN {X 160.99, Y 176.37, Z 0.00, A 0, B 0, C 0} C_DIS
LIN {X 161.09, Y 176.08, Z 0.00, A 0, B 0, C 0} C_DIS
LIN {X 161.15, Y 175.77, Z 0.00, A 0, B 0, C 0} C_DIS
LIN {X 161.21, Y 175.45, Z 0.00, A 0, B 0, C 0} C_DIS
LIN {X 161.28, Y 175.14, Z 0.00, A 0, B 0, C 0} C_DIS
LIN {X 161.37, Y 174.84, Z 0.00, A 0, B 0, C 0} C_DIS
LIN {X 161.45, Y 174.54, Z 0.00, A 0, B 0, C 0} C_DIS
LIN {X 161.52, Y 174.23, Z 0.00, A 0, B 0, C 0} C_DIS
LIN {X 161.58, Y 173.91, Z 0.00, A 0, B 0, C 0} C_DIS
LIN {X 161.63, Y 173.60, Z 0.00, A 0, B 0, C 0} C_DIS
LIN {X 161.68, Y 173.28, Z 0.00, A 0, B 0, C 0} C_DIS
LIN {X 161.73, Y 172.96, Z 0.00, A 0, B 0, C 0} C_DIS
LIN {X 161.78, Y 172.64, Z 0.00, A 0, B 0, C 0} C_DIS
LIN {X 161.83, Y 172.32, Z 0.00, A 0, B 0, C 0} C_DIS
LIN {X 161.88, Y 172.00, Z 0.00, A 0, B 0, C 0} C_DIS
LIN {X 161.94, Y 171.68, Z 0.00, A 0, B 0, C 0} C_DIS
LIN {X 162.00, Y 171.37, Z 0.00, A 0, B 0, C 0} C_DIS
LIN {X 162.05, Y 171.05, Z 0.00, A 0, B 0, C 0} C_DIS
LIN {X 162.10, Y 170.73, Z 0.00, A 0, B 0, C 0} C_DIS
LIN {X 162.15, Y 170.41, Z 0.00, A 0, B 0, C 0} C_DIS
LIN {X 162.18, Y 170.09, Z 0.00, A 0, B 0, C 0} C_DIS
LIN {X 162.22, Y 169.77, Z 0.00, A 0, B 0, C 0} C_DIS
LIN {X 162.24, Y 169.44, Z 0.00, A 0, B 0, C 0} C_DIS
LIN {X 162.27, Y 169.12, Z 0.00, A 0, B 0, C 0} C_DIS
LIN {X 162.31, Y 168.79, Z 0.00, A 0, B 0, C 0} C_DIS
LIN {X 162.35, Y 168.47, Z 0.00, A 0, B 0, C 0} C_DIS
LIN {X 162.41, Y 168.16, Z 0.00, A 0, B 0, C 0} C_DIS
LIN {X 162.47, Y 167.84, Z 0.00, A 0, B 0, C 0} C_DIS
LIN {X 162.53, Y 167.53, Z 0.00, A 0, B 0, C 0} C_DIS
LIN {X 162.58, Y 167.21, Z 0.00, A 0, B 0, C 0} C_DIS
LIN {X 162.62, Y 166.88, Z 0.00, A 0, B 0, C 0} C_DIS
LIN {X 162.64, Y 166.56, Z 0.00, A 0, B 0, C 0} C_DIS
LIN {X 162.66, Y 166.23, Z 0.00, A 0, B 0, C 0} C_DIS
LIN {X 162.67, Y 165.91, Z 0.00, A 0, B 0, C 0} C_DIS
LIN {X 162.67, Y 165.58, Z 0.00, A 0, B 0, C 0} C_DIS
LIN {X 162.67, Y 165.25, Z 0.00, A 0, B 0, C 0} C_DIS
LIN {X 162.66, Y 164.92, Z 0.00, A 0, B 0, C 0} C_DIS
LIN {X 162.65, Y 164.59, Z 0.00, A 0, B 0, C 0} C_DIS
LIN {X 162.65, Y 164.26, Z 0.00, A 0, B 0, C 0} C_DIS
LIN {X 162.65, Y 163.94, Z 0.00, A 0, B 0, C 0} C_DIS
LIN {X 162.67, Y 163.61, Z 0.00, A 0, B 0, C 0} C_DIS
LIN {X 162.70, Y 163.29, Z 0.00, A 0, B 0, C 0} C_DIS
LIN {X 162.74, Y 162.97, Z 0.00, A 0, B 0, C 0} C_DIS
LIN {X 162.78, Y 162.65, Z 0.00, A 0, B 0, C 0} C_DIS
LIN {X 162.84, Y 162.33, Z 0.00, A 0, B 0, C 0} C_DIS
LIN {X 162.89, Y 162.01, Z 0.00, A 0, B 0, C 0} C_DIS
LIN {X 162.94, Y 161.69, Z 0.00, A 0, B 0, C 0} C_DIS
LIN {X 162.99, Y 161.37, Z 0.00, A 0, B 0, C 0} C_DIS
LIN {X 163.04, Y 161.06, Z 0.00, A 0, B 0, C 0} C_DIS
LIN {X 163.08, Y 160.73, Z 0.00, A 0, B 0, C 0} C_DIS
LIN {X 163.10, Y 160.41, Z 0.00, A 0, B 0, C 0} C_DIS
LIN {X 163.11, Y 160.08, Z 0.00, A 0, B 0, C 0} C_DIS
LIN {X 163.12, Y 159.75, Z 0.00, A 0, B 0, C 0} C_DIS
LIN {X 163.11, Y 159.42, Z 0.00, A 0, B 0, C 0} C_DIS
LIN {X 163.09, Y 159.10, Z 0.00, A 0, B 0, C 0} C_DIS
LIN {X 163.06, Y 158.77, Z 0.00, A 0, B 0, C 0} C_DIS
LIN {X 163.02, Y 158.45, Z 0.00, A 0, B 0, C 0} C_DIS
LIN {X 162.98, Y 158.13, Z 0.00, A 0, B 0, C 0} C_DIS
LIN {X 162.93, Y 157.81, Z 0.00, A 0, B 0, C 0} C_DIS
LIN {X 162.87, Y 157.50, Z 0.00, A 0, B 0, C 0} C_DIS
LIN {X 162.81, Y 157.18, Z 0.00, A 0, B 0, C 0} C_DIS
LIN {X 162.75, Y 156.86, Z 0.00, A 0, B 0, C 0} C_DIS
LIN {X 162.71, Y 156.54, Z 0.00, A 0, B 0, C 0} C_DIS
LIN {X 162.68, Y 156.22, Z 0.00, A 0, B 0, C 0} C_DIS
LIN {X 162.66, Y 155.89, Z 0.00, A 0, B 0, C 0} C_DIS
LIN {X 162.66, Y 155.56, Z 0.00, A 0, B 0, C 0} C_DIS
LIN {X 162.66, Y 155.24, Z 0.00, A 0, B 0, C 0} C_DIS
LIN {X 162.67, Y 154.91, Z 0.00, A 0, B 0, C 0} C_DIS
LIN {X 162.67, Y 154.58, Z 0.00, A 0, B 0, C 0} C_DIS
LIN {X 162.67, Y 154.25, Z 0.00, A 0, B 0, C 0} C_DIS
LIN {X 162.67, Y 153.92, Z 0.00, A 0, B 0, C 0} C_DIS
LIN {X 162.66, Y 153.60, Z 0.00, A 0, B 0, C 0} C_DIS
LIN {X 162.65, Y 153.27, Z 0.00, A 0, B 0, C 0} C_DIS
LIN {X 162.62, Y 152.95, Z 0.00, A 0, B 0, C 0} C_DIS
LIN {X 162.59, Y 152.62, Z 0.00, A 0, B 0, C 0} C_DIS
LIN {X 162.56, Y 152.30, Z 0.00, A 0, B 0, C 0} C_DIS
LIN {X 162.51, Y 151.98, Z 0.00, A 0, B 0, C 0} C_DIS
LIN {X 162.46, Y 151.66, Z 0.00, A 0, B 0, C 0} C_DIS
LIN {X 162.40, Y 151.35, Z 0.00, A 0, B 0, C 0} C_DIS
LIN {X 162.34, Y 151.03, Z 0.00, A 0, B 0, C 0} C_DIS
LIN {X 162.29, Y 150.71, Z 0.00, A 0, B 0, C 0} C_DIS
LIN {X 162.23, Y 150.39, Z 0.00, A 0, B 0, C 0} C_DIS
LIN {X 162.17, Y 150.08, Z 0.00, A 0, B 0, C 0} C_DIS
LIN {X 162.12, Y 149.76, Z 0.00, A 0, B 0, C 0} C_DIS
LIN {X 162.07, Y 149.44, Z 0.00, A 0, B 0, C 0} C_DIS
LIN {X 162.02, Y 149.12, Z 0.00, A 0, B 0, C 0} C_DIS
LIN {X 161.97, Y 148.81, Z 0.00, A 0, B 0, C 0} C_DIS
LIN {X 161.92, Y 148.49, Z 0.00, A 0, B 0, C 0} C_DIS
LIN {X 161.87, Y 148.17, Z 0.00, A 0, B 0, C 0} C_DIS
LIN {X 161.82, Y 147.85, Z 0.00, A 0, B 0, C 0} C_DIS
LIN {X 161.76, Y 147.53, Z 0.00, A 0, B 0, C 0} C_DIS
LIN {X 161.71, Y 147.21, Z 0.00, A 0, B 0, C 0} C_DIS
LIN {X 161.66, Y 146.89, Z 0.00, A 0, B 0, C 0} C_DIS
LIN {X 161.60, Y 146.58, Z 0.00, A 0, B 0, C 0} C_DIS
LIN {X 161.54, Y 146.26, Z 0.00, A 0, B 0, C 0} C_DIS
LIN {X 161.48, Y 145.95, Z 0.00, A 0, B 0, C 0} C_DIS
LIN {X 161.42, Y 145.64, Z 0.00, A 0, B 0, C 0} C_DIS
LIN {X 161.34, Y 145.34, Z 0.00, A 0, B 0, C 0} C_DIS
LIN {X 161.25, Y 145.04, Z 0.00, A 0, B 0, C 0} C_DIS
LIN {X 161.18, Y 144.72, Z 0.00, A 0, B 0, C 0} C_DIS
LIN {X 161.13, Y 144.41, Z 0.00, A 0, B 0, C 0} C_DIS
LIN {X 161.05, Y 144.10, Z 0.00, A 0, B 0, C 0} C_DIS
LIN {X 160.94, Y 143.82, Z 0.00, A 0, B 0, C 0} C_DIS
LIN {X 160.82, Y 143.54, Z 0.00, A 0, B 0, C 0} C_DIS
LIN {X 160.73, Y 143.25, Z 0.00, A 0, B 0, C 0} C_DIS
LIN {X 160.67, Y 142.93, Z 0.00, A 0, B 0, C 0} C_DIS
LIN {X 160.62, Y 142.61, Z 0.00, A 0, B 0, C 0} C_DIS
LIN {X 160.53, Y 142.31, Z 0.00, A 0, B 0, C 0} C_DIS
LIN {X 160.44, Y 142.02, Z 0.00, A 0, B 0, C 0} C_DIS
LIN {X 160.37, Y 141.70, Z 0.00, A 0, B 0, C 0} C_DIS
LIN {X 160.31, Y 141.39, Z 0.00, A 0, B 0, C 0} C_DIS
LIN {X 160.24, Y 141.08, Z 0.00, A 0, B 0, C 0} C_DIS
LIN {X 160.15, Y 140.78, Z 0.00, A 0, B 0, C 0} C_DIS
LIN {X 160.05, Y 140.50, Z 0.00, A 0, B 0, C 0} C_DIS
LIN {X 159.94, Y 140.22, Z 0.00, A 0, B 0, C 0} C_DIS
LIN {X 159.82, Y 139.94, Z 0.00, A 0, B 0, C 0} C_DIS
LIN {X 159.69, Y 139.67, Z 0.00, A 0, B 0, C 0} C_DIS
LIN {X 159.56, Y 139.41, Z 0.00, A 0, B 0, C 0} C_DIS
LIN {X 159.44, Y 139.14, Z 0.00, A 0, B 0, C 0} C_DIS
LIN {X 159.32, Y 138.87, Z 0.00, A 0, B 0, C 0} C_DIS
LIN {X 159.20, Y 138.59, Z 0.00, A 0, B 0, C 0} C_DIS
LIN {X 159.10, Y 138.30, Z 0.00, A 0, B 0, C 0} C_DIS
LIN {X 159.01, Y 138.01, Z 0.00, A 0, B 0, C 0} C_DIS
LIN {X 158.92, Y 137.71, Z 0.00, A 0, B 0, C 0} C_DIS
LIN {X 158.82, Y 137.42, Z 0.00, A 0, B 0, C 0} C_DIS
LIN {X 158.71, Y 137.14, Z 0.00, A 0, B 0, C 0} C_DIS
LIN {X 158.59, Y 136.86, Z 0.00, A 0, B 0, C 0} C_DIS
LIN {X 158.47, Y 136.59, Z 0.00, A 0, B 0, C 0} C_DIS
LIN {X 158.35, Y 136.32, Z 0.00, A 0, B 0, C 0} C_DIS
LIN {X 158.23, Y 136.05, Z 0.00, A 0, B 0, C 0} C_DIS
LIN {X 158.11, Y 135.77, Z 0.00, A 0, B 0, C 0} C_DIS
LIN {X 157.98, Y 135.50, Z 0.00, A 0, B 0, C 0} C_DIS
LIN {X 157.86, Y 135.23, Z 0.00, A 0, B 0, C 0} C_DIS
LIN {X 157.74, Y 134.96, Z 0.00, A 0, B 0, C 0} C_DIS
LIN {X 157.62, Y 134.68, Z 0.00, A 0, B 0, C 0} C_DIS
LIN {X 157.50, Y 134.41, Z 0.00, A 0, B 0, C 0} C_DIS
LIN {X 157.38, Y 134.14, Z 0.00, A 0, B 0, C 0} C_DIS
LIN {X 157.26, Y 133.86, Z 0.00, A 0, B 0, C 0} C_DIS
LIN {X 157.14, Y 133.59, Z 0.00, A 0, B 0, C 0} C_DIS
LIN {X 157.02, Y 133.32, Z 0.00, A 0, B 0, C 0} C_DIS
LIN {X 156.90, Y 133.04, Z 0.00, A 0, B 0, C 0} C_DIS
LIN {X 156.78, Y 132.77, Z 0.00, A 0, B 0, C 0} C_DIS
LIN {X 156.65, Y 132.51, Z 0.00, A 0, B 0, C 0} C_DIS
LIN {X 156.53, Y 132.24, Z 0.00, A 0, B 0, C 0} C_DIS
LIN {X 156.39, Y 131.99, Z 0.00, A 0, B 0, C 0} C_DIS
LIN {X 156.23, Y 131.76, Z 0.00, A 0, B 0, C 0} C_DIS
LIN {X 156.07, Y 131.54, Z 0.00, A 0, B 0, C 0} C_DIS
LIN {X 155.91, Y 131.32, Z 0.00, A 0, B 0, C 0} C_DIS
LIN {X 155.76, Y 131.08, Z 0.00, A 0, B 0, C 0} C_DIS
LIN {X 155.63, Y 130.82, Z 0.00, A 0, B 0, C 0} C_DIS
LIN {X 155.50, Y 130.55, Z 0.00, A 0, B 0, C 0} C_DIS
LIN {X 155.38, Y 130.28, Z 0.00, A 0, B 0, C 0} C_DIS
LIN {X 155.26, Y 130.01, Z 0.00, A 0, B 0, C 0} C_DIS
LIN {X 155.15, Y 129.73, Z 0.00, A 0, B 0, C 0} C_DIS
LIN {X 155.03, Y 129.46, Z 0.00, A 0, B 0, C 0} C_DIS
LIN {X 154.90, Y 129.19, Z 0.00, A 0, B 0, C 0} C_DIS
LIN {X 154.77, Y 128.93, Z 0.00, A 0, B 0, C 0} C_DIS
LIN {X 154.62, Y 128.69, Z 0.00, A 0, B 0, C 0} C_DIS
LIN {X 154.47, Y 128.46, Z 0.00, A 0, B 0, C 0} C_DIS
LIN {X 154.31, Y 128.23, Z 0.00, A 0, B 0, C 0} C_DIS
LIN {X 154.16, Y 128.00, Z 0.00, A 0, B 0, C 0} C_DIS
LIN {X 154.00, Y 127.77, Z 0.00, A 0, B 0, C 0} C_DIS
LIN {X 153.85, Y 127.54, Z 0.00, A 0, B 0, C 0} C_DIS
LIN {X 153.69, Y 127.31, Z 0.00, A 0, B 0, C 0} C_DIS
LIN {X 153.54, Y 127.07, Z 0.00, A 0, B 0, C 0} C_DIS
LIN {X 153.39, Y 126.84, Z 0.00, A 0, B 0, C 0} C_DIS
LIN {X 153.23, Y 126.61, Z 0.00, A 0, B 0, C 0} C_DIS
LIN {X 153.08, Y 126.38, Z 0.00, A 0, B 0, C 0} C_DIS
LIN {X 152.93, Y 126.15, Z 0.00, A 0, B 0, C 0} C_DIS
LIN {X 152.77, Y 125.91, Z 0.00, A 0, B 0, C 0} C_DIS
LIN {X 152.62, Y 125.68, Z 0.00, A 0, B 0, C 0} C_DIS
LIN {X 152.47, Y 125.45, Z 0.00, A 0, B 0, C 0} C_DIS
LIN {X 152.31, Y 125.22, Z 0.00, A 0, B 0, C 0} C_DIS
LIN {X 152.16, Y 124.99, Z 0.00, A 0, B 0, C 0} C_DIS
LIN {X 152.00, Y 124.76, Z 0.00, A 0, B 0, C 0} C_DIS
LIN {X 151.85, Y 124.53, Z 0.00, A 0, B 0, C 0} C_DIS
LIN {X 151.70, Y 124.30, Z 0.00, A 0, B 0, C 0} C_DIS
LIN {X 151.54, Y 124.06, Z 0.00, A 0, B 0, C 0} C_DIS
LIN {X 151.39, Y 123.83, Z 0.00, A 0, B 0, C 0} C_DIS
LIN {X 151.24, Y 123.59, Z 0.00, A 0, B 0, C 0} C_DIS
LIN {X 151.09, Y 123.36, Z 0.00, A 0, B 0, C 0} C_DIS
LIN {X 150.93, Y 123.13, Z 0.00, A 0, B 0, C 0} C_DIS
LIN {X 150.77, Y 122.91, Z 0.00, A 0, B 0, C 0} C_DIS
LIN {X 150.61, Y 122.70, Z 0.00, A 0, B 0, C 0} C_DIS
LIN {X 150.43, Y 122.50, Z 0.00, A 0, B 0, C 0} C_DIS
LIN {X 150.25, Y 122.32, Z 0.00, A 0, B 0, C 0} C_DIS
LIN {X 150.07, Y 122.14, Z 0.00, A 0, B 0, C 0} C_DIS
LIN {X 149.89, Y 121.96, Z 0.00, A 0, B 0, C 0} C_DIS
LIN {X 149.70, Y 121.78, Z 0.00, A 0, B 0, C 0} C_DIS
LIN {X 149.52, Y 121.60, Z 0.00, A 0, B 0, C 0} C_DIS
LIN {X 149.35, Y 121.40, Z 0.00, A 0, B 0, C 0} C_DIS
LIN {X 149.19, Y 121.19, Z 0.00, A 0, B 0, C 0} C_DIS
LIN {X 149.04, Y 120.95, Z 0.00, A 0, B 0, C 0} C_DIS
LIN {X 148.89, Y 120.71, Z 0.00, A 0, B 0, C 0} C_DIS
LIN {X 148.74, Y 120.47, Z 0.00, A 0, B 0, C 0} C_DIS
LIN {X 148.58, Y 120.25, Z 0.00, A 0, B 0, C 0} C_DIS
LIN {X 148.41, Y 120.05, Z 0.00, A 0, B 0, C 0} C_DIS
LIN {X 148.23, Y 119.86, Z 0.00, A 0, B 0, C 0} C_DIS
LIN {X 148.06, Y 119.67, Z 0.00, A 0, B 0, C 0} C_DIS
LIN {X 147.88, Y 119.49, Z 0.00, A 0, B 0, C 0} C_DIS
LIN {X 147.69, Y 119.31, Z 0.00, A 0, B 0, C 0} C_DIS
LIN {X 147.50, Y 119.14, Z 0.00, A 0, B 0, C 0} C_DIS
LIN {X 147.32, Y 118.96, Z 0.00, A 0, B 0, C 0} C_DIS
LIN {X 147.15, Y 118.76, Z 0.00, A 0, B 0, C 0} C_DIS
LIN {X 147.00, Y 118.52, Z 0.00, A 0, B 0, C 0} C_DIS
LIN {X 146.88, Y 118.26, Z 0.00, A 0, B 0, C 0} C_DIS
LIN {X 146.77, Y 117.97, Z 0.00, A 0, B 0, C 0} C_DIS
LIN {X 146.69, Y 117.67, Z 0.00, A 0, B 0, C 0} C_DIS
LIN {X 146.63, Y 117.35, Z 0.00, A 0, B 0, C 0} C_DIS
LIN {X 146.59, Y 117.03, Z 0.00, A 0, B 0, C 0} C_DIS
LIN {X 146.57, Y 116.70, Z 0.00, A 0, B 0, C 0} C_DIS
LIN {X 146.56, Y 116.37, Z 0.00, A 0, B 0, C 0} C_DIS
LIN {X 146.56, Y 116.05, Z 0.00, A 0, B 0, C 0} C_DIS
LIN {X 146.57, Y 115.72, Z 0.00, A 0, B 0, C 0} C_DIS
LIN {X 146.57, Y 115.39, Z 0.00, A 0, B 0, C 0} C_DIS
LIN {X 146.58, Y 115.06, Z 0.00, A 0, B 0, C 0} C_DIS
LIN {X 146.58, Y 114.73, Z 0.00, A 0, B 0, C 0} C_DIS
LIN {X 146.57, Y 114.41, Z 0.00, A 0, B 0, C 0} C_DIS
LIN {X 146.57, Y 114.08, Z 0.00, A 0, B 0, C 0} C_DIS
LIN {X 146.57, Y 113.75, Z 0.00, A 0, B 0, C 0} C_DIS
LIN {X 146.57, Y 113.42, Z 0.00, A 0, B 0, C 0} C_DIS
LIN {X 146.57, Y 113.10, Z 0.00, A 0, B 0, C 0} C_DIS
LIN {X 146.57, Y 112.77, Z 0.00, A 0, B 0, C 0} C_DIS
LIN {X 146.57, Y 112.44, Z 0.00, A 0, B 0, C 0} C_DIS
LIN {X 146.57, Y 112.11, Z 0.00, A 0, B 0, C 0} C_DIS
LIN {X 146.57, Y 111.78, Z 0.00, A 0, B 0, C 0} C_DIS
LIN {X 146.57, Y 111.46, Z 0.00, A 0, B 0, C 0} C_DIS
LIN {X 146.57, Y 111.13, Z 0.00, A 0, B 0, C 0} C_DIS
LIN {X 146.57, Y 110.80, Z 0.00, A 0, B 0, C 0} C_DIS
LIN {X 146.57, Y 110.47, Z 0.00, A 0, B 0, C 0} C_DIS
LIN {X 146.57, Y 110.15, Z 0.00, A 0, B 0, C 0} C_DIS
LIN {X 146.57, Y 109.82, Z 0.00, A 0, B 0, C 0} C_DIS
LIN {X 146.57, Y 109.49, Z 0.00, A 0, B 0, C 0} C_DIS
LIN {X 146.57, Y 109.16, Z 0.00, A 0, B 0, C 0} C_DIS
LIN {X 146.57, Y 108.83, Z 0.00, A 0, B 0, C 0} C_DIS
LIN {X 146.57, Y 108.51, Z 0.00, A 0, B 0, C 0} C_DIS
LIN {X 146.57, Y 108.18, Z 0.00, A 0, B 0, C 0} C_DIS
LIN {X 146.57, Y 107.85, Z 0.00, A 0, B 0, C 0} C_DIS
LIN {X 146.57, Y 107.52, Z 0.00, A 0, B 0, C 0} C_DIS
LIN {X 146.57, Y 107.20, Z 0.00, A 0, B 0, C 0} C_DIS
LIN {X 146.57, Y 106.87, Z 0.00, A 0, B 0, C 0} C_DIS
LIN {X 146.57, Y 106.54, Z 0.00, A 0, B 0, C 0} C_DIS
LIN {X 146.57, Y 106.21, Z 0.00, A 0, B 0, C 0} C_DIS
LIN {X 146.57, Y 105.89, Z 0.00, A 0, B 0, C 0} C_DIS
LIN {X 146.57, Y 105.56, Z 0.00, A 0, B 0, C 0} C_DIS
LIN {X 146.57, Y 105.23, Z 0.00, A 0, B 0, C 0} C_DIS
LIN {X 146.57, Y 104.90, Z 0.00, A 0, B 0, C 0} C_DIS
LIN {X 146.57, Y 104.57, Z 0.00, A 0, B 0, C 0} C_DIS
LIN {X 146.57, Y 104.25, Z 0.00, A 0, B 0, C 0} C_DIS
LIN {X 146.57, Y 103.92, Z 0.00, A 0, B 0, C 0} C_DIS
LIN {X 146.57, Y 103.59, Z 0.00, A 0, B 0, C 0} C_DIS
LIN {X 146.57, Y 103.26, Z 0.00, A 0, B 0, C 0} C_DIS
LIN {X 146.57, Y 102.94, Z 0.00, A 0, B 0, C 0} C_DIS
LIN {X 146.57, Y 102.61, Z 0.00, A 0, B 0, C 0} C_DIS
LIN {X 146.57, Y 102.28, Z 0.00, A 0, B 0, C 0} C_DIS
LIN {X 146.57, Y 101.95, Z 0.00, A 0, B 0, C 0} C_DIS
LIN {X 146.57, Y 101.62, Z 0.00, A 0, B 0, C 0} C_DIS
LIN {X 146.57, Y 101.30, Z 0.00, A 0, B 0, C 0} C_DIS
LIN {X 146.57, Y 100.97, Z 0.00, A 0, B 0, C 0} C_DIS
LIN {X 146.57, Y 100.64, Z 0.00, A 0, B 0, C 0} C_DIS
LIN {X 146.57, Y 100.31, Z 0.00, A 0, B 0, C 0} C_DIS
LIN {X 146.57, Y 99.99, Z 0.00, A 0, B 0, C 0} C_DIS
LIN {X 146.57, Y 99.66, Z 0.00, A 0, B 0, C 0} C_DIS
LIN {X 146.57, Y 99.33, Z 0.00, A 0, B 0, C 0} C_DIS
LIN {X 146.57, Y 99.00, Z 0.00, A 0, B 0, C 0} C_DIS
LIN {X 146.57, Y 98.68, Z 0.00, A 0, B 0, C 0} C_DIS
LIN {X 146.57, Y 98.35, Z 0.00, A 0, B 0, C 0} C_DIS
LIN {X 146.57, Y 98.02, Z 0.00, A 0, B 0, C 0} C_DIS
LIN {X 146.57, Y 97.69, Z 0.00, A 0, B 0, C 0} C_DIS
LIN {X 146.57, Y 97.36, Z 0.00, A 0, B 0, C 0} C_DIS
LIN {X 146.57, Y 97.04, Z 0.00, A 0, B 0, C 0} C_DIS
LIN {X 146.57, Y 96.71, Z 0.00, A 0, B 0, C 0} C_DIS
LIN {X 146.57, Y 96.38, Z 0.00, A 0, B 0, C 0} C_DIS
LIN {X 146.57, Y 96.05, Z 0.00, A 0, B 0, C 0} C_DIS
LIN {X 146.57, Y 95.73, Z 0.00, A 0, B 0, C 0} C_DIS
LIN {X 146.57, Y 95.40, Z 0.00, A 0, B 0, C 0} C_DIS
LIN {X 146.57, Y 95.07, Z 0.00, A 0, B 0, C 0} C_DIS
LIN {X 146.57, Y 94.74, Z 0.00, A 0, B 0, C 0} C_DIS
LIN {X 146.57, Y 94.42, Z 0.00, A 0, B 0, C 0} C_DIS
LIN {X 146.57, Y 94.09, Z 0.00, A 0, B 0, C 0} C_DIS
LIN {X 146.57, Y 93.76, Z 0.00, A 0, B 0, C 0} C_DIS
LIN {X 146.57, Y 93.43, Z 0.00, A 0, B 0, C 0} C_DIS
LIN {X 146.57, Y 93.10, Z 0.00, A 0, B 0, C 0} C_DIS
LIN {X 146.57, Y 92.78, Z 0.00, A 0, B 0, C 0} C_DIS
LIN {X 146.57, Y 92.45, Z 0.00, A 0, B 0, C 0} C_DIS
LIN {X 146.57, Y 92.12, Z 0.00, A 0, B 0, C 0} C_DIS
LIN {X 146.57, Y 91.79, Z 0.00, A 0, B 0, C 0} C_DIS
LIN {X 146.57, Y 91.47, Z 0.00, A 0, B 0, C 0} C_DIS
LIN {X 146.57, Y 91.14, Z 0.00, A 0, B 0, C 0} C_DIS
LIN {X 146.57, Y 90.81, Z 0.00, A 0, B 0, C 0} C_DIS
LIN {X 146.57, Y 90.48, Z 0.00, A 0, B 0, C 0} C_DIS
LIN {X 146.57, Y 90.15, Z 0.00, A 0, B 0, C 0} C_DIS
LIN {X 146.57, Y 89.83, Z 0.00, A 0, B 0, C 0} C_DIS
LIN {X 146.57, Y 89.50, Z 0.00, A 0, B 0, C 0} C_DIS
LIN {X 146.57, Y 89.17, Z 0.00, A 0, B 0, C 0} C_DIS
LIN {X 146.57, Y 88.84, Z 0.00, A 0, B 0, C 0} C_DIS
LIN {X 146.57, Y 88.52, Z 0.00, A 0, B 0, C 0} C_DIS
LIN {X 146.57, Y 88.19, Z 0.00, A 0, B 0, C 0} C_DIS
LIN {X 146.57, Y 87.86, Z 0.00, A 0, B 0, C 0} C_DIS
LIN {X 146.57, Y 87.53, Z 0.00, A 0, B 0, C 0} C_DIS
LIN {X 146.57, Y 87.21, Z 0.00, A 0, B 0, C 0} C_DIS
LIN {X 146.57, Y 86.88, Z 0.00, A 0, B 0, C 0} C_DIS
LIN {X 146.57, Y 86.55, Z 0.00, A 0, B 0, C 0} C_DIS
LIN {X 146.57, Y 86.22, Z 0.00, A 0, B 0, C 0} C_DIS
LIN {X 146.57, Y 85.90, Z 0.00, A 0, B 0, C 0} C_DIS
LIN {X 146.57, Y 85.57, Z 0.00, A 0, B 0, C 0} C_DIS
LIN {X 146.58, Y 85.24, Z 0.00, A 0, B 0, C 0} C_DIS
LIN {X 146.58, Y 84.91, Z 0.00, A 0, B 0, C 0} C_DIS
LIN {X 146.58, Y 84.58, Z 0.00, A 0, B 0, C 0} C_DIS
LIN {X 146.58, Y 84.25, Z 0.00, A 0, B 0, C 0} C_DIS
LIN {X 146.58, Y 83.93, Z 0.00, A 0, B 0, C 0} C_DIS
LIN {X 146.57, Y 83.60, Z 0.00, A 0, B 0, C 0} C_DIS
LIN {X 146.56, Y 83.27, Z 0.00, A 0, B 0, C 0} C_DIS
LIN {X 146.54, Y 82.95, Z 0.00, A 0, B 0, C 0} C_DIS
LIN {X 146.52, Y 82.63, Z 0.00, A 0, B 0, C 0} C_DIS
LIN {X 146.49, Y 82.30, Z 0.00, A 0, B 0, C 0} C_DIS
LIN {X 146.44, Y 81.98, Z 0.00, A 0, B 0, C 0} C_DIS
LIN {X 146.39, Y 81.66, Z 0.00, A 0, B 0, C 0} C_DIS
LIN {X 146.31, Y 81.35, Z 0.00, A 0, B 0, C 0} C_DIS
LIN {X 146.21, Y 81.06, Z 0.00, A 0, B 0, C 0} C_DIS
LIN {X 146.10, Y 80.78, Z 0.00, A 0, B 0, C 0} C_DIS
LIN {X 145.99, Y 80.50, Z 0.00, A 0, B 0, C 0} C_DIS
LIN {X 145.87, Y 80.23, Z 0.00, A 0, B 0, C 0} C_DIS
LIN {X 145.74, Y 79.96, Z 0.00, A 0, B 0, C 0} C_DIS
LIN {X 145.60, Y 79.71, Z 0.00, A 0, B 0, C 0} C_DIS
LIN {X 145.45, Y 79.48, Z 0.00, A 0, B 0, C 0} C_DIS
LIN {X 145.29, Y 79.25, Z 0.00, A 0, B 0, C 0} C_DIS
LIN {X 145.14, Y 79.02, Z 0.00, A 0, B 0, C 0} C_DIS
LIN {X 144.99, Y 78.78, Z 0.00, A 0, B 0, C 0} C_DIS
LIN {X 144.84, Y 78.54, Z 0.00, A 0, B 0, C 0} C_DIS
LIN {X 144.68, Y 78.32, Z 0.00, A 0, B 0, C 0} C_DIS
LIN {X 144.51, Y 78.12, Z 0.00, A 0, B 0, C 0} C_DIS
LIN {X 144.33, Y 77.93, Z 0.00, A 0, B 0, C 0} C_DIS
LIN {X 144.16, Y 77.73, Z 0.00, A 0, B 0, C 0} C_DIS
LIN {X 143.99, Y 77.53, Z 0.00, A 0, B 0, C 0} C_DIS
LIN {X 143.82, Y 77.32, Z 0.00, A 0, B 0, C 0} C_DIS
LIN {X 143.67, Y 77.09, Z 0.00, A 0, B 0, C 0} C_DIS
LIN {X 143.52, Y 76.84, Z 0.00, A 0, B 0, C 0} C_DIS
LIN {X 143.39, Y 76.59, Z 0.00, A 0, B 0, C 0} C_DIS
LIN {X 143.26, Y 76.32, Z 0.00, A 0, B 0, C 0} C_DIS
LIN {X 143.13, Y 76.06, Z 0.00, A 0, B 0, C 0} C_DIS
LIN {X 143.00, Y 75.80, Z 0.00, A 0, B 0, C 0} C_DIS
LIN {X 142.86, Y 75.56, Z 0.00, A 0, B 0, C 0} C_DIS
LIN {X 142.70, Y 75.33, Z 0.00, A 0, B 0, C 0} C_DIS
LIN {X 142.54, Y 75.11, Z 0.00, A 0, B 0, C 0} C_DIS
LIN {X 142.38, Y 74.88, Z 0.00, A 0, B 0, C 0} C_DIS
LIN {X 142.24, Y 74.64, Z 0.00, A 0, B 0, C 0} C_DIS
LIN {X 142.11, Y 74.38, Z 0.00, A 0, B 0, C 0} C_DIS
LIN {X 141.98, Y 74.11, Z 0.00, A 0, B 0, C 0} C_DIS
LIN {X 141.87, Y 73.83, Z 0.00, A 0, B 0, C 0} C_DIS
LIN {X 141.75, Y 73.55, Z 0.00, A 0, B 0, C 0} C_DIS
LIN {X 141.63, Y 73.28, Z 0.00, A 0, B 0, C 0} C_DIS
LIN {X 141.51, Y 73.01, Z 0.00, A 0, B 0, C 0} C_DIS
LIN {X 141.38, Y 72.74, Z 0.00, A 0, B 0, C 0} C_DIS
LIN {X 141.26, Y 72.47, Z 0.00, A 0, B 0, C 0} C_DIS
LIN {X 141.13, Y 72.20, Z 0.00, A 0, B 0, C 0} C_DIS
LIN {X 141.02, Y 71.93, Z 0.00, A 0, B 0, C 0} C_DIS
LIN {X 140.90, Y 71.65, Z 0.00, A 0, B 0, C 0} C_DIS
LIN {X 140.80, Y 71.36, Z 0.00, A 0, B 0, C 0} C_DIS
LIN {X 140.71, Y 71.06, Z 0.00, A 0, B 0, C 0} C_DIS
LIN {X 140.62, Y 70.77, Z 0.00, A 0, B 0, C 0} C_DIS
LIN {X 140.52, Y 70.48, Z 0.00, A 0, B 0, C 0} C_DIS
LIN {X 140.41, Y 70.20, Z 0.00, A 0, B 0, C 0} C_DIS
LIN {X 140.31, Y 69.90, Z 0.00, A 0, B 0, C 0} C_DIS
LIN {X 140.23, Y 69.60, Z 0.00, A 0, B 0, C 0} C_DIS
LIN {X 140.14, Y 69.30, Z 0.00, A 0, B 0, C 0} C_DIS
LIN {X 140.03, Y 69.02, Z 0.00, A 0, B 0, C 0} C_DIS
LIN {X 139.92, Y 68.74, Z 0.00, A 0, B 0, C 0} C_DIS
LIN {X 139.83, Y 68.44, Z 0.00, A 0, B 0, C 0} C_DIS
LIN {X 139.76, Y 68.13, Z 0.00, A 0, B 0, C 0} C_DIS
LIN {X 139.65, Y 67.84, Z 0.00, A 0, B 0, C 0} C_DIS
LIN {X 139.53, Y 67.57, Z 0.00, A 0, B 0, C 0} C_DIS
LIN {X 139.44, Y 67.28, Z 0.00, A 0, B 0, C 0} C_DIS
LIN {X 139.37, Y 66.97, Z 0.00, A 0, B 0, C 0} C_DIS
LIN {X 139.32, Y 66.65, Z 0.00, A 0, B 0, C 0} C_DIS
LIN {X 139.24, Y 66.34, Z 0.00, A 0, B 0, C 0} C_DIS
LIN {X 139.15, Y 66.04, Z 0.00, A 0, B 0, C 0} C_DIS
LIN {X 139.07, Y 65.74, Z 0.00, A 0, B 0, C 0} C_DIS
LIN {X 139.00, Y 65.43, Z 0.00, A 0, B 0, C 0} C_DIS
LIN {X 138.95, Y 65.11, Z 0.00, A 0, B 0, C 0} C_DIS
LIN {X 138.90, Y 64.79, Z 0.00, A 0, B 0, C 0} C_DIS
LIN {X 138.84, Y 64.48, Z 0.00, A 0, B 0, C 0} C_DIS
LIN {X 138.75, Y 64.18, Z 0.00, A 0, B 0, C 0} C_DIS
LIN {X 138.66, Y 63.88, Z 0.00, A 0, B 0, C 0} C_DIS
LIN {X 138.59, Y 63.57, Z 0.00, A 0, B 0, C 0} C_DIS
LIN {X 138.53, Y 63.26, Z 0.00, A 0, B 0, C 0} C_DIS
LIN {X 138.48, Y 62.94, Z 0.00, A 0, B 0, C 0} C_DIS
LIN {X 138.43, Y 62.62, Z 0.00, A 0, B 0, C 0} C_DIS
LIN {X 138.38, Y 62.29, Z 0.00, A 0, B 0, C 0} C_DIS
LIN {X 138.34, Y 61.97, Z 0.00, A 0, B 0, C 0} C_DIS
LIN {X 138.33, Y 61.65, Z 0.00, A 0, B 0, C 0} C_DIS
LIN {X 138.39, Y 61.34, Z 0.00, A 0, B 0, C 0} C_DIS
LIN {X 138.51, Y 61.05, Z 0.00, A 0, B 0, C 0} C_DIS
LIN {X 138.67, Y 60.83, Z 0.00, A 0, B 0, C 0} C_DIS
LIN {X 138.86, Y 60.69, Z 0.00, A 0, B 0, C 0} C_DIS
LIN {X 139.08, Y 60.62, Z 0.00, A 0, B 0, C 0} C_DIS
LIN {X 139.29, Y 60.59, Z 0.00, A 0, B 0, C 0} C_DIS
LIN {X 139.51, Y 60.59, Z 0.00, A 0, B 0, C 0} C_DIS
LIN {X 139.73, Y 60.59, Z 0.00, A 0, B 0, C 0} C_DIS
LIN {X 139.95, Y 60.59, Z 0.00, A 0, B 0, C 0} C_DIS
LIN {X 140.16, Y 60.59, Z 0.00, A 0, B 0, C 0} C_DIS
LIN {X 140.38, Y 60.59, Z 0.00, A 0, B 0, C 0} C_DIS
LIN {X 140.60, Y 60.59, Z 0.00, A 0, B 0, C 0} C_DIS
LIN {X 140.82, Y 60.59, Z 0.00, A 0, B 0, C 0} C_DIS
LIN {X 141.03, Y 60.59, Z 0.00, A 0, B 0, C 0} C_DIS
LIN {X 141.25, Y 60.59, Z 0.00, A 0, B 0, C 0} C_DIS
LIN {X 141.47, Y 60.59, Z 0.00, A 0, B 0, C 0} C_DIS
LIN {X 141.69, Y 60.59, Z 0.00, A 0, B 0, C 0} C_DIS
LIN {X 141.90, Y 60.59, Z 0.00, A 0, B 0, C 0} C_DIS
LIN {X 142.12, Y 60.59, Z 0.00, A 0, B 0, C 0} C_DIS
LIN {X 142.34, Y 60.59, Z 0.00, A 0, B 0, C 0} C_DIS
LIN {X 142.56, Y 60.59, Z 0.00, A 0, B 0, C 0} C_DIS
LIN {X 142.77, Y 60.59, Z 0.00, A 0, B 0, C 0} C_DIS
LIN {X 142.99, Y 60.59, Z 0.00, A 0, B 0, C 0} C_DIS
LIN {X 143.21, Y 60.59, Z 0.00, A 0, B 0, C 0} C_DIS
LIN {X 143.42, Y 60.59, Z 0.00, A 0, B 0, C 0} C_DIS
LIN {X 143.64, Y 60.59, Z 0.00, A 0, B 0, C 0} C_DIS
LIN {X 143.86, Y 60.59, Z 0.00, A 0, B 0, C 0} C_DIS
LIN {X 144.08, Y 60.59, Z 0.00, A 0, B 0, C 0} C_DIS
LIN {X 144.29, Y 60.59, Z 0.00, A 0, B 0, C 0} C_DIS
LIN {X 144.51, Y 60.59, Z 0.00, A 0, B 0, C 0} C_DIS
LIN {X 144.73, Y 60.59, Z 0.00, A 0, B 0, C 0} C_DIS
LIN {X 144.95, Y 60.59, Z 0.00, A 0, B 0, C 0} C_DIS
LIN {X 145.17, Y 60.59, Z 0.00, A 0, B 0, C 0} C_DIS
LIN {X 145.38, Y 60.59, Z 0.00, A 0, B 0, C 0} C_DIS
LIN {X 145.60, Y 60.59, Z 0.00, A 0, B 0, C 0} C_DIS
LIN {X 145.82, Y 60.59, Z 0.00, A 0, B 0, C 0} C_DIS
LIN {X 146.04, Y 60.59, Z 0.00, A 0, B 0, C 0} C_DIS
LIN {X 146.25, Y 60.59, Z 0.00, A 0, B 0, C 0} C_DIS
LIN {X 146.47, Y 60.59, Z 0.00, A 0, B 0, C 0} C_DIS
LIN {X 146.68, Y 60.60, Z 0.00, A 0, B 0, C 0} C_DIS
LIN {X 146.90, Y 60.61, Z 0.00, A 0, B 0, C 0} C_DIS
LIN {X 147.12, Y 60.64, Z 0.00, A 0, B 0, C 0} C_DIS
LIN {X 147.34, Y 60.70, Z 0.00, A 0, B 0, C 0} C_DIS
LIN {X 147.56, Y 60.79, Z 0.00, A 0, B 0, C 0} C_DIS
LIN {X 147.75, Y 60.94, Z 0.00, A 0, B 0, C 0} C_DIS
LIN {X 147.90, Y 61.15, Z 0.00, A 0, B 0, C 0} C_DIS
LIN {X 148.01, Y 61.42, Z 0.00, A 0, B 0, C 0} C_DIS
LIN {X 148.11, Y 61.72, Z 0.00, A 0, B 0, C 0} C_DIS
LIN {X 148.20, Y 62.02, Z 0.00, A 0, B 0, C 0} C_DIS
LIN {X 148.28, Y 62.32, Z 0.00, A 0, B 0, C 0} C_DIS
LIN {X 148.35, Y 62.63, Z 0.00, A 0, B 0, C 0} C_DIS
LIN {X 148.41, Y 62.95, Z 0.00, A 0, B 0, C 0} C_DIS
LIN {X 148.48, Y 63.26, Z 0.00, A 0, B 0, C 0} C_DIS
LIN {X 148.57, Y 63.55, Z 0.00, A 0, B 0, C 0} C_DIS
LIN {X 148.68, Y 63.84, Z 0.00, A 0, B 0, C 0} C_DIS
LIN {X 148.79, Y 64.11, Z 0.00, A 0, B 0, C 0} C_DIS
LIN {X 148.92, Y 64.39, Z 0.00, A 0, B 0, C 0} C_DIS
LIN {X 149.04, Y 64.65, Z 0.00, A 0, B 0, C 0} C_DIS
LIN {X 149.16, Y 64.92, Z 0.00, A 0, B 0, C 0} C_DIS
LIN {X 149.29, Y 65.20, Z 0.00, A 0, B 0, C 0} C_DIS
LIN {X 149.40, Y 65.47, Z 0.00, A 0, B 0, C 0} C_DIS
LIN {X 149.52, Y 65.75, Z 0.00, A 0, B 0, C 0} C_DIS
LIN {X 149.64, Y 66.02, Z 0.00, A 0, B 0, C 0} C_DIS
LIN {X 149.76, Y 66.29, Z 0.00, A 0, B 0, C 0} C_DIS
LIN {X 149.89, Y 66.56, Z 0.00, A 0, B 0, C 0} C_DIS
LIN {X 150.02, Y 66.82, Z 0.00, A 0, B 0, C 0} C_DIS
LIN {X 150.16, Y 67.06, Z 0.00, A 0, B 0, C 0} C_DIS
LIN {X 150.31, Y 67.30, Z 0.00, A 0, B 0, C 0} C_DIS
LIN {X 150.47, Y 67.52, Z 0.00, A 0, B 0, C 0} C_DIS
LIN {X 150.63, Y 67.75, Z 0.00, A 0, B 0, C 0} C_DIS
LIN {X 150.79, Y 67.98, Z 0.00, A 0, B 0, C 0} C_DIS
LIN {X 150.93, Y 68.22, Z 0.00, A 0, B 0, C 0} C_DIS
LIN {X 151.08, Y 68.46, Z 0.00, A 0, B 0, C 0} C_DIS
LIN {X 151.24, Y 68.69, Z 0.00, A 0, B 0, C 0} C_DIS
LIN {X 151.40, Y 68.91, Z 0.00, A 0, B 0, C 0} C_DIS
LIN {X 151.56, Y 69.12, Z 0.00, A 0, B 0, C 0} C_DIS
LIN {X 151.74, Y 69.32, Z 0.00, A 0, B 0, C 0} C_DIS
LIN {X 151.91, Y 69.51, Z 0.00, A 0, B 0, C 0} C_DIS
LIN {X 152.10, Y 69.68, Z 0.00, A 0, B 0, C 0} C_DIS
LIN {X 152.28, Y 69.86, Z 0.00, A 0, B 0, C 0} C_DIS
LIN {X 152.46, Y 70.04, Z 0.00, A 0, B 0, C 0} C_DIS
LIN {X 152.65, Y 70.22, Z 0.00, A 0, B 0, C 0} C_DIS
LIN {X 152.82, Y 70.40, Z 0.00, A 0, B 0, C 0} C_DIS
LIN {X 153.00, Y 70.59, Z 0.00, A 0, B 0, C 0} C_DIS
LIN {X 153.18, Y 70.77, Z 0.00, A 0, B 0, C 0} C_DIS
LIN {X 153.36, Y 70.95, Z 0.00, A 0, B 0, C 0} C_DIS
LIN {X 153.55, Y 71.13, Z 0.00, A 0, B 0, C 0} C_DIS
LIN {X 153.74, Y 71.29, Z 0.00, A 0, B 0, C 0} C_DIS
LIN {X 153.94, Y 71.40, Z 0.00, A 0, B 0, C 0} C_DIS
LIN {X 154.15, Y 71.48, Z 0.00, A 0, B 0, C 0} C_DIS
LIN {X 154.36, Y 71.58, Z 0.00, A 0, B 0, C 0} C_DIS
LIN {X 154.56, Y 71.71, Z 0.00, A 0, B 0, C 0} C_DIS
LIN {X 154.76, Y 71.85, Z 0.00, A 0, B 0, C 0} C_DIS
LIN {X 154.96, Y 71.96, Z 0.00, A 0, B 0, C 0} C_DIS
LIN {X 155.17, Y 72.04, Z 0.00, A 0, B 0, C 0} C_DIS
LIN {X 155.39, Y 72.11, Z 0.00, A 0, B 0, C 0} C_DIS
LIN {X 155.59, Y 72.20, Z 0.00, A 0, B 0, C 0} C_DIS
LIN {X 155.80, Y 72.32, Z 0.00, A 0, B 0, C 0} C_DIS
LIN {X 156.00, Y 72.45, Z 0.00, A 0, B 0, C 0} C_DIS
LIN {X 156.20, Y 72.57, Z 0.00, A 0, B 0, C 0} C_DIS
LIN {X 156.40, Y 72.67, Z 0.00, A 0, B 0, C 0} C_DIS
LIN {X 156.61, Y 72.75, Z 0.00, A 0, B 0, C 0} C_DIS
LIN {X 156.83, Y 72.83, Z 0.00, A 0, B 0, C 0} C_DIS
LIN {X 157.04, Y 72.89, Z 0.00, A 0, B 0, C 0} C_DIS
LIN {X 157.25, Y 72.96, Z 0.00, A 0, B 0, C 0} C_DIS
LIN {X 157.47, Y 73.01, Z 0.00, A 0, B 0, C 0} C_DIS
LIN {X 157.68, Y 73.05, Z 0.00, A 0, B 0, C 0} C_DIS
LIN {X 157.90, Y 73.06, Z 0.00, A 0, B 0, C 0} C_DIS
LIN {X 158.12, Y 73.06, Z 0.00, A 0, B 0, C 0} C_DIS
LIN {X 158.33, Y 73.05, Z 0.00, A 0, B 0, C 0} C_DIS
LIN {X 158.55, Y 73.05, Z 0.00, A 0, B 0, C 0} C_DIS
LIN {X 158.77, Y 73.04, Z 0.00, A 0, B 0, C 0} C_DIS
LIN {X 158.99, Y 73.04, Z 0.00, A 0, B 0, C 0} C_DIS
LIN {X 159.20, Y 73.04, Z 0.00, A 0, B 0, C 0} C_DIS
LIN {X 159.42, Y 73.04, Z 0.00, A 0, B 0, C 0} C_DIS
LIN {X 159.64, Y 73.04, Z 0.00, A 0, B 0, C 0} C_DIS
LIN {X 159.86, Y 73.04, Z 0.00, A 0, B 0, C 0} C_DIS
LIN {X 160.07, Y 73.04, Z 0.00, A 0, B 0, C 0} C_DIS
LIN {X 160.29, Y 73.04, Z 0.00, A 0, B 0, C 0} C_DIS
LIN {X 160.51, Y 73.04, Z 0.00, A 0, B 0, C 0} C_DIS
LIN {X 160.73, Y 73.04, Z 0.00, A 0, B 0, C 0} C_DIS
LIN {X 160.94, Y 73.04, Z 0.00, A 0, B 0, C 0} C_DIS
LIN {X 161.16, Y 73.04, Z 0.00, A 0, B 0, C 0} C_DIS
LIN {X 161.38, Y 73.04, Z 0.00, A 0, B 0, C 0} C_DIS
LIN {X 161.60, Y 73.04, Z 0.00, A 0, B 0, C 0} C_DIS
LIN {X 161.81, Y 73.04, Z 0.00, A 0, B 0, C 0} C_DIS
LIN {X 162.03, Y 73.04, Z 0.00, A 0, B 0, C 0} C_DIS
LIN {X 162.25, Y 73.04, Z 0.00, A 0, B 0, C 0} C_DIS
LIN {X 162.47, Y 73.04, Z 0.00, A 0, B 0, C 0} C_DIS
LIN {X 162.68, Y 73.04, Z 0.00, A 0, B 0, C 0} C_DIS
LIN {X 162.90, Y 73.04, Z 0.00, A 0, B 0, C 0} C_DIS
LIN {X 163.12, Y 73.04, Z 0.00, A 0, B 0, C 0} C_DIS
LIN {X 163.34, Y 73.04, Z 0.00, A 0, B 0, C 0} C_DIS
LIN {X 163.55, Y 73.04, Z 0.00, A 0, B 0, C 0} C_DIS
LIN {X 163.77, Y 73.04, Z 0.00, A 0, B 0, C 0} C_DIS
LIN {X 163.99, Y 73.04, Z 0.00, A 0, B 0, C 0} C_DIS
LIN {X 164.21, Y 73.04, Z 0.00, A 0, B 0, C 0} C_DIS
LIN {X 164.42, Y 73.04, Z 0.00, A 0, B 0, C 0} C_DIS
LIN {X 164.64, Y 73.04, Z 0.00, A 0, B 0, C 0} C_DIS
LIN {X 164.86, Y 73.04, Z 0.00, A 0, B 0, C 0} C_DIS
LIN {X 165.08, Y 73.04, Z 0.00, A 0, B 0, C 0} C_DIS
LIN {X 165.29, Y 73.04, Z 0.00, A 0, B 0, C 0} C_DIS
LIN {X 165.51, Y 73.04, Z 0.00, A 0, B 0, C 0} C_DIS
LIN {X 165.73, Y 73.04, Z 0.00, A 0, B 0, C 0} C_DIS
LIN {X 165.95, Y 73.04, Z 0.00, A 0, B 0, C 0} C_DIS
LIN {X 166.16, Y 73.04, Z 0.00, A 0, B 0, C 0} C_DIS
LIN {X 166.38, Y 73.04, Z 0.00, A 0, B 0, C 0} C_DIS
LIN {X 166.60, Y 73.04, Z 0.00, A 0, B 0, C 0} C_DIS
LIN {X 166.81, Y 73.04, Z 0.00, A 0, B 0, C 0} C_DIS
LIN {X 167.03, Y 73.04, Z 0.00, A 0, B 0, C 0} C_DIS
LIN {X 167.25, Y 73.04, Z 0.00, A 0, B 0, C 0} C_DIS
LIN {X 167.47, Y 73.04, Z 0.00, A 0, B 0, C 0} C_DIS
LIN {X 167.68, Y 73.04, Z 0.00, A 0, B 0, C 0} C_DIS
LIN {X 167.90, Y 73.04, Z 0.00, A 0, B 0, C 0} C_DIS
LIN {X 168.12, Y 73.04, Z 0.00, A 0, B 0, C 0} C_DIS
LIN {X 168.34, Y 73.04, Z 0.00, A 0, B 0, C 0} C_DIS
LIN {X 168.55, Y 73.04, Z 0.00, A 0, B 0, C 0} C_DIS
LIN {X 168.77, Y 73.04, Z 0.00, A 0, B 0, C 0} C_DIS
LIN {X 168.99, Y 73.04, Z 0.00, A 0, B 0, C 0} C_DIS
LIN {X 169.21, Y 73.04, Z 0.00, A 0, B 0, C 0} C_DIS
LIN {X 169.42, Y 73.04, Z 0.00, A 0, B 0, C 0} C_DIS
LIN {X 169.64, Y 73.04, Z 0.00, A 0, B 0, C 0} C_DIS
LIN {X 169.86, Y 73.04, Z 0.00, A 0, B 0, C 0} C_DIS
LIN {X 170.08, Y 73.04, Z 0.00, A 0, B 0, C 0} C_DIS
LIN {X 170.29, Y 73.04, Z 0.00, A 0, B 0, C 0} C_DIS
LIN {X 170.51, Y 73.04, Z 0.00, A 0, B 0, C 0} C_DIS
LIN {X 170.73, Y 73.04, Z 0.00, A 0, B 0, C 0} C_DIS
LIN {X 170.95, Y 73.04, Z 0.00, A 0, B 0, C 0} C_DIS
LIN {X 171.16, Y 73.04, Z 0.00, A 0, B 0, C 0} C_DIS
LIN {X 171.38, Y 73.04, Z 0.00, A 0, B 0, C 0} C_DIS
LIN {X 171.60, Y 73.04, Z 0.00, A 0, B 0, C 0} C_DIS
LIN {X 171.82, Y 73.04, Z 0.00, A 0, B 0, C 0} C_DIS
LIN {X 172.03, Y 73.04, Z 0.00, A 0, B 0, C 0} C_DIS
LIN {X 172.25, Y 73.04, Z 0.00, A 0, B 0, C 0} C_DIS
LIN {X 172.47, Y 73.04, Z 0.00, A 0, B 0, C 0} C_DIS
LIN {X 172.69, Y 73.04, Z 0.00, A 0, B 0, C 0} C_DIS
LIN {X 172.90, Y 73.04, Z 0.00, A 0, B 0, C 0} C_DIS
LIN {X 173.12, Y 73.04, Z 0.00, A 0, B 0, C 0} C_DIS
LIN {X 173.34, Y 73.04, Z 0.00, A 0, B 0, C 0} C_DIS
LIN {X 173.56, Y 73.04, Z 0.00, A 0, B 0, C 0} C_DIS
LIN {X 173.77, Y 73.04, Z 0.00, A 0, B 0, C 0} C_DIS
LIN {X 173.99, Y 73.04, Z 0.00, A 0, B 0, C 0} C_DIS
LIN {X 174.21, Y 73.04, Z 0.00, A 0, B 0, C 0} C_DIS
LIN {X 174.43, Y 73.04, Z 0.00, A 0, B 0, C 0} C_DIS
LIN {X 174.64, Y 73.04, Z 0.00, A 0, B 0, C 0} C_DIS
LIN {X 174.86, Y 73.04, Z 0.00, A 0, B 0, C 0} C_DIS
LIN {X 175.08, Y 73.04, Z 0.00, A 0, B 0, C 0} C_DIS
LIN {X 175.30, Y 73.05, Z 0.00, A 0, B 0, C 0} C_DIS
LIN {X 175.51, Y 73.05, Z 0.00, A 0, B 0, C 0} C_DIS
LIN {X 175.73, Y 73.05, Z 0.00, A 0, B 0, C 0} C_DIS
LIN {X 175.95, Y 73.05, Z 0.00, A 0, B 0, C 0} C_DIS
LIN {X 176.17, Y 73.05, Z 0.00, A 0, B 0, C 0} C_DIS
LIN {X 176.38, Y 73.05, Z 0.00, A 0, B 0, C 0} C_DIS
LIN {X 176.60, Y 73.05, Z 0.00, A 0, B 0, C 0} C_DIS
LIN {X 176.82, Y 73.05, Z 0.00, A 0, B 0, C 0} C_DIS
LIN {X 177.04, Y 73.05, Z 0.00, A 0, B 0, C 0} C_DIS
LIN {X 177.25, Y 73.04, Z 0.00, A 0, B 0, C 0} C_DIS
LIN {X 177.47, Y 73.04, Z 0.00, A 0, B 0, C 0} C_DIS
LIN {X 177.69, Y 73.04, Z 0.00, A 0, B 0, C 0} C_DIS
LIN {X 177.90, Y 73.04, Z 0.00, A 0, B 0, C 0} C_DIS
LIN {X 178.12, Y 73.04, Z 0.00, A 0, B 0, C 0} C_DIS
LIN {X 178.34, Y 73.04, Z 0.00, A 0, B 0, C 0} C_DIS
LIN {X 178.56, Y 73.04, Z 0.00, A 0, B 0, C 0} C_DIS
LIN {X 178.77, Y 73.04, Z 0.00, A 0, B 0, C 0} C_DIS
LIN {X 178.99, Y 73.04, Z 0.00, A 0, B 0, C 0} C_DIS
LIN {X 179.21, Y 73.04, Z 0.00, A 0, B 0, C 0} C_DIS
LIN {X 179.43, Y 73.04, Z 0.00, A 0, B 0, C 0} C_DIS
LIN {X 179.64, Y 73.04, Z 0.00, A 0, B 0, C 0} C_DIS
LIN {X 179.86, Y 73.04, Z 0.00, A 0, B 0, C 0} C_DIS
LIN {X 180.08, Y 73.05, Z 0.00, A 0, B 0, C 0} C_DIS
LIN {X 180.30, Y 73.05, Z 0.00, A 0, B 0, C 0} C_DIS
LIN {X 180.52, Y 73.05, Z 0.00, A 0, B 0, C 0} C_DIS
LIN {X 180.73, Y 73.06, Z 0.00, A 0, B 0, C 0} C_DIS
LIN {X 180.95, Y 73.06, Z 0.00, A 0, B 0, C 0} C_DIS
LIN {X 181.17, Y 73.05, Z 0.00, A 0, B 0, C 0} C_DIS
LIN {X 181.39, Y 73.03, Z 0.00, A 0, B 0, C 0} C_DIS
LIN {X 181.60, Y 73.01, Z 0.00, A 0, B 0, C 0} C_DIS
LIN {X 181.82, Y 72.98, Z 0.00, A 0, B 0, C 0} C_DIS
LIN {X 182.03, Y 72.93, Z 0.00, A 0, B 0, C 0} C_DIS
LIN {X 182.24, Y 72.86, Z 0.00, A 0, B 0, C 0} C_DIS
LIN {X 182.45, Y 72.79, Z 0.00, A 0, B 0, C 0} C_DIS
LIN {X 182.66, Y 72.71, Z 0.00, A 0, B 0, C 0} C_DIS
LIN {X 182.87, Y 72.62, Z 0.00, A 0, B 0, C 0} C_DIS
LIN {X 183.08, Y 72.53, Z 0.00, A 0, B 0, C 0} C_DIS
LIN {X 183.30, Y 72.45, Z 0.00, A 0, B 0, C 0} C_DIS
LIN {X 183.51, Y 72.36, Z 0.00, A 0, B 0, C 0} C_DIS
LIN {X 183.72, Y 72.28, Z 0.00, A 0, B 0, C 0} C_DIS
LIN {X 183.93, Y 72.21, Z 0.00, A 0, B 0, C 0} C_DIS
LIN {X 184.14, Y 72.14, Z 0.00, A 0, B 0, C 0} C_DIS
LIN {X 184.35, Y 72.07, Z 0.00, A 0, B 0, C 0} C_DIS
LIN {X 184.56, Y 71.98, Z 0.00, A 0, B 0, C 0} C_DIS
LIN {X 184.77, Y 71.88, Z 0.00, A 0, B 0, C 0} C_DIS
LIN {X 184.97, Y 71.76, Z 0.00, A 0, B 0, C 0} C_DIS
LIN {X 185.17, Y 71.62, Z 0.00, A 0, B 0, C 0} C_DIS
LIN {X 185.37, Y 71.50, Z 0.00, A 0, B 0, C 0} C_DIS
LIN {X 185.59, Y 71.44, Z 0.00, A 0, B 0, C 0} C_DIS
LIN {X 185.79, Y 71.34, Z 0.00, A 0, B 0, C 0} C_DIS
LIN {X 185.98, Y 71.17, Z 0.00, A 0, B 0, C 0} C_DIS
LIN {X 186.17, Y 71.00, Z 0.00, A 0, B 0, C 0} C_DIS
LIN {X 186.36, Y 70.85, Z 0.00, A 0, B 0, C 0} C_DIS
LIN {X 186.56, Y 70.74, Z 0.00, A 0, B 0, C 0} C_DIS
LIN {X 186.77, Y 70.65, Z 0.00, A 0, B 0, C 0} C_DIS
LIN {X 186.98, Y 70.55, Z 0.00, A 0, B 0, C 0} C_DIS
LIN {X 187.18, Y 70.42, Z 0.00, A 0, B 0, C 0} C_DIS
LIN {X 187.38, Y 70.30, Z 0.00, A 0, B 0, C 0} C_DIS
LIN {X 187.58, Y 70.19, Z 0.00, A 0, B 0, C 0} C_DIS
LIN {X 187.79, Y 70.09, Z 0.00, A 0, B 0, C 0} C_DIS
LIN {X 188.00, Y 69.99, Z 0.00, A 0, B 0, C 0} C_DIS
LIN {X 188.19, Y 69.85, Z 0.00, A 0, B 0, C 0} C_DIS
LIN {X 188.38, Y 69.69, Z 0.00, A 0, B 0, C 0} C_DIS
LIN {X 188.57, Y 69.52, Z 0.00, A 0, B 0, C 0} C_DIS
LIN {X 188.76, Y 69.38, Z 0.00, A 0, B 0, C 0} C_DIS
LIN {X 188.96, Y 69.24, Z 0.00, A 0, B 0, C 0} C_DIS
LIN {X 189.15, Y 69.09, Z 0.00, A 0, B 0, C 0} C_DIS
LIN {X 189.34, Y 68.93, Z 0.00, A 0, B 0, C 0} C_DIS
LIN {X 189.52, Y 68.75, Z 0.00, A 0, B 0, C 0} C_DIS
LIN {X 189.70, Y 68.57, Z 0.00, A 0, B 0, C 0} C_DIS
LIN {X 189.88, Y 68.38, Z 0.00, A 0, B 0, C 0} C_DIS
LIN {X 190.06, Y 68.19, Z 0.00, A 0, B 0, C 0} C_DIS
LIN {X 190.24, Y 68.00, Z 0.00, A 0, B 0, C 0} C_DIS
LIN {X 190.42, Y 67.82, Z 0.00, A 0, B 0, C 0} C_DIS
LIN {X 190.60, Y 67.64, Z 0.00, A 0, B 0, C 0} C_DIS
LIN {X 190.78, Y 67.45, Z 0.00, A 0, B 0, C 0} C_DIS
LIN {X 190.96, Y 67.28, Z 0.00, A 0, B 0, C 0} C_DIS
LIN {X 191.14, Y 67.10, Z 0.00, A 0, B 0, C 0} C_DIS
LIN {X 191.33, Y 66.92, Z 0.00, A 0, B 0, C 0} C_DIS
LIN {X 191.51, Y 66.74, Z 0.00, A 0, B 0, C 0} C_DIS
LIN {X 191.69, Y 66.56, Z 0.00, A 0, B 0, C 0} C_DIS
LIN {X 191.87, Y 66.38, Z 0.00, A 0, B 0, C 0} C_DIS
LIN {X 192.05, Y 66.20, Z 0.00, A 0, B 0, C 0} C_DIS
LIN {X 192.23, Y 66.00, Z 0.00, A 0, B 0, C 0} C_DIS
LIN {X 192.40, Y 65.80, Z 0.00, A 0, B 0, C 0} C_DIS
LIN {X 192.56, Y 65.59, Z 0.00, A 0, B 0, C 0} C_DIS
LIN {X 192.72, Y 65.37, Z 0.00, A 0, B 0, C 0} C_DIS
LIN {X 192.88, Y 65.15, Z 0.00, A 0, B 0, C 0} C_DIS
LIN {X 193.03, Y 64.91, Z 0.00, A 0, B 0, C 0} C_DIS
LIN {X 193.18, Y 64.68, Z 0.00, A 0, B 0, C 0} C_DIS
LIN {X 193.34, Y 64.44, Z 0.00, A 0, B 0, C 0} C_DIS
LIN {X 193.49, Y 64.21, Z 0.00, A 0, B 0, C 0} C_DIS
LIN {X 193.64, Y 63.97, Z 0.00, A 0, B 0, C 0} C_DIS
LIN {X 193.79, Y 63.74, Z 0.00, A 0, B 0, C 0} C_DIS
LIN {X 193.95, Y 63.51, Z 0.00, A 0, B 0, C 0} C_DIS
LIN {X 194.10, Y 63.28, Z 0.00, A 0, B 0, C 0} C_DIS
LIN {X 194.26, Y 63.05, Z 0.00, A 0, B 0, C 0} C_DIS
LIN {X 194.41, Y 62.82, Z 0.00, A 0, B 0, C 0} C_DIS
LIN {X 194.57, Y 62.59, Z 0.00, A 0, B 0, C 0} C_DIS
LIN {X 194.72, Y 62.36, Z 0.00, A 0, B 0, C 0} C_DIS
LIN {X 194.87, Y 62.12, Z 0.00, A 0, B 0, C 0} C_DIS
LIN {X 195.03, Y 61.89, Z 0.00, A 0, B 0, C 0} C_DIS
LIN {X 195.18, Y 61.66, Z 0.00, A 0, B 0, C 0} C_DIS
LIN {X 195.33, Y 61.43, Z 0.00, A 0, B 0, C 0} C_DIS
LIN {X 195.49, Y 61.20, Z 0.00, A 0, B 0, C 0} C_DIS
LIN {X 195.65, Y 60.97, Z 0.00, A 0, B 0, C 0} C_DIS
LIN {X 195.80, Y 60.74, Z 0.00, A 0, B 0, C 0} C_DIS
LIN {X 195.95, Y 60.50, Z 0.00, A 0, B 0, C 0} C_DIS
LIN {X 196.09, Y 60.26, Z 0.00, A 0, B 0, C 0} C_DIS
LIN {X 196.23, Y 60.00, Z 0.00, A 0, B 0, C 0} C_DIS
LIN {X 196.36, Y 59.74, Z 0.00, A 0, B 0, C 0} C_DIS
LIN {X 196.48, Y 59.47, Z 0.00, A 0, B 0, C 0} C_DIS
LIN {X 196.60, Y 59.20, Z 0.00, A 0, B 0, C 0} C_DIS
LIN {X 196.72, Y 58.92, Z 0.00, A 0, B 0, C 0} C_DIS
LIN {X 196.83, Y 58.64, Z 0.00, A 0, B 0, C 0} C_DIS
LIN {X 196.95, Y 58.37, Z 0.00, A 0, B 0, C 0} C_DIS
LIN {X 197.07, Y 58.09, Z 0.00, A 0, B 0, C 0} C_DIS
LIN {X 197.20, Y 57.82, Z 0.00, A 0, B 0, C 0} C_DIS
LIN {X 197.32, Y 57.55, Z 0.00, A 0, B 0, C 0} C_DIS
LIN {X 197.43, Y 57.28, Z 0.00, A 0, B 0, C 0} C_DIS
LIN {X 197.54, Y 57.00, Z 0.00, A 0, B 0, C 0} C_DIS
LIN {X 197.64, Y 56.71, Z 0.00, A 0, B 0, C 0} C_DIS
LIN {X 197.73, Y 56.41, Z 0.00, A 0, B 0, C 0} C_DIS
LIN {X 197.82, Y 56.11, Z 0.00, A 0, B 0, C 0} C_DIS
LIN {X 197.92, Y 55.82, Z 0.00, A 0, B 0, C 0} C_DIS
LIN {X 198.05, Y 55.55, Z 0.00, A 0, B 0, C 0} C_DIS
LIN {X 198.18, Y 55.29, Z 0.00, A 0, B 0, C 0} C_DIS
LIN {X 198.30, Y 55.02, Z 0.00, A 0, B 0, C 0} C_DIS
LIN {X 198.42, Y 54.74, Z 0.00, A 0, B 0, C 0} C_DIS
LIN {X 198.54, Y 54.46, Z 0.00, A 0, B 0, C 0} C_DIS
LIN {X 198.66, Y 54.19, Z 0.00, A 0, B 0, C 0} C_DIS
LIN {X 198.78, Y 53.92, Z 0.00, A 0, B 0, C 0} C_DIS
LIN {X 198.88, Y 53.63, Z 0.00, A 0, B 0, C 0} C_DIS
LIN {X 198.97, Y 53.34, Z 0.00, A 0, B 0, C 0} C_DIS
LIN {X 199.06, Y 53.04, Z 0.00, A 0, B 0, C 0} C_DIS
LIN {X 199.16, Y 52.75, Z 0.00, A 0, B 0, C 0} C_DIS
LIN {X 199.27, Y 52.46, Z 0.00, A 0, B 0, C 0} C_DIS
LIN {X 199.39, Y 52.19, Z 0.00, A 0, B 0, C 0} C_DIS
LIN {X 199.51, Y 51.92, Z 0.00, A 0, B 0, C 0} C_DIS
LIN {X 199.64, Y 51.65, Z 0.00, A 0, B 0, C 0} C_DIS
LIN {X 199.76, Y 51.38, Z 0.00, A 0, B 0, C 0} C_DIS
LIN {X 199.89, Y 51.11, Z 0.00, A 0, B 0, C 0} C_DIS
LIN {X 200.00, Y 50.84, Z 0.00, A 0, B 0, C 0} C_DIS
LIN {X 200.11, Y 50.56, Z 0.00, A 0, B 0, C 0} C_DIS
LIN {X 200.21, Y 50.27, Z 0.00, A 0, B 0, C 0} C_DIS
LIN {X 200.30, Y 49.96, Z 0.00, A 0, B 0, C 0} C_DIS
LIN {X 200.38, Y 49.66, Z 0.00, A 0, B 0, C 0} C_DIS
LIN {X 200.49, Y 49.38, Z 0.00, A 0, B 0, C 0} C_DIS
LIN {X 200.61, Y 49.10, Z 0.00, A 0, B 0, C 0} C_DIS
LIN {X 200.70, Y 48.80, Z 0.00, A 0, B 0, C 0} C_DIS
LIN {X 200.73, Y 48.49, Z 0.00, A 0, B 0, C 0} C_DIS
LIN {X 200.74, Y 48.16, Z 0.00, A 0, B 0, C 0} C_DIS
LIN {X 200.75, Y 47.82, Z 0.00, A 0, B 0, C 0} C_DIS
LIN {X 200.73, Y 47.49, Z 0.00, A 0, B 0, C 0} C_DIS
LIN {X 200.66, Y 47.19, Z 0.00, A 0, B 0, C 0} C_DIS
LIN {X 200.54, Y 46.92, Z 0.00, A 0, B 0, C 0} C_DIS
LIN {X 200.40, Y 46.67, Z 0.00, A 0, B 0, C 0} C_DIS
LIN {X 200.25, Y 46.43, Z 0.00, A 0, B 0, C 0} C_DIS
LIN {X 200.10, Y 46.20, Z 0.00, A 0, B 0, C 0} C_DIS
LIN {X 199.93, Y 45.98, Z 0.00, A 0, B 0, C 0} C_DIS
LIN {X 199.76, Y 45.79, Z 0.00, A 0, B 0, C 0} C_DIS
LIN {X 199.58, Y 45.61, Z 0.00, A 0, B 0, C 0} C_DIS
LIN {X 199.40, Y 45.41, Z 0.00, A 0, B 0, C 0} C_DIS
LIN {X 199.24, Y 45.20, Z 0.00, A 0, B 0, C 0} C_DIS
LIN {X 199.09, Y 44.97, Z 0.00, A 0, B 0, C 0} C_DIS
LIN {X 198.93, Y 44.73, Z 0.00, A 0, B 0, C 0} C_DIS
LIN {X 198.79, Y 44.49, Z 0.00, A 0, B 0, C 0} C_DIS
LIN {X 198.65, Y 44.24, Z 0.00, A 0, B 0, C 0} C_DIS
LIN {X 198.53, Y 43.97, Z 0.00, A 0, B 0, C 0} C_DIS
LIN {X 198.41, Y 43.70, Z 0.00, A 0, B 0, C 0} C_DIS
LIN {X 198.29, Y 43.42, Z 0.00, A 0, B 0, C 0} C_DIS
LIN {X 198.18, Y 43.14, Z 0.00, A 0, B 0, C 0} C_DIS
LIN {X 198.06, Y 42.87, Z 0.00, A 0, B 0, C 0} C_DIS
LIN {X 197.93, Y 42.59, Z 0.00, A 0, B 0, C 0} C_DIS
LIN {X 197.81, Y 42.33, Z 0.00, A 0, B 0, C 0} C_DIS
LIN {X 197.68, Y 42.06, Z 0.00, A 0, B 0, C 0} C_DIS
LIN {X 197.56, Y 41.79, Z 0.00, A 0, B 0, C 0} C_DIS
LIN {X 197.45, Y 41.51, Z 0.00, A 0, B 0, C 0} C_DIS
LIN {X 197.34, Y 41.22, Z 0.00, A 0, B 0, C 0} C_DIS
LIN {X 197.26, Y 40.92, Z 0.00, A 0, B 0, C 0} C_DIS
LIN {X 197.17, Y 40.62, Z 0.00, A 0, B 0, C 0} C_DIS
LIN {X 197.06, Y 40.34, Z 0.00, A 0, B 0, C 0} C_DIS
LIN {X 196.95, Y 40.06, Z 0.00, A 0, B 0, C 0} C_DIS
LIN {X 196.86, Y 39.77, Z 0.00, A 0, B 0, C 0} C_DIS
LIN {X 196.78, Y 39.46, Z 0.00, A 0, B 0, C 0} C_DIS
LIN {X 196.69, Y 39.16, Z 0.00, A 0, B 0, C 0} C_DIS
LIN {X 196.56, Y 38.90, Z 0.00, A 0, B 0, C 0} C_DIS
LIN {X 196.40, Y 38.68, Z 0.00, A 0, B 0, C 0} C_DIS
LIN {X 196.24, Y 38.44, Z 0.00, A 0, B 0, C 0} C_DIS
LIN {X 196.10, Y 38.20, Z 0.00, A 0, B 0, C 0} C_DIS
LIN {X 195.92, Y 38.01, Z 0.00, A 0, B 0, C 0} C_DIS
LIN {X 195.72, Y 37.88, Z 0.00, A 0, B 0, C 0} C_DIS
LIN {X 195.52, Y 37.77, Z 0.00, A 0, B 0, C 0} C_DIS
LIN {X 195.33, Y 37.62, Z 0.00, A 0, B 0, C 0} C_DIS
LIN {X 195.14, Y 37.44, Z 0.00, A 0, B 0, C 0} C_DIS
LIN {X 194.95, Y 37.28, Z 0.00, A 0, B 0, C 0} C_DIS
LIN {X 194.75, Y 37.17, Z 0.00, A 0, B 0, C 0} C_DIS
LIN {X 194.54, Y 37.09, Z 0.00, A 0, B 0, C 0} C_DIS
LIN {X 194.32, Y 37.02, Z 0.00, A 0, B 0, C 0} C_DIS
LIN {X 194.11, Y 36.95, Z 0.00, A 0, B 0, C 0} C_DIS
LIN {X 193.90, Y 36.89, Z 0.00, A 0, B 0, C 0} C_DIS
LIN {X 193.68, Y 36.86, Z 0.00, A 0, B 0, C 0} C_DIS
LIN {X 193.47, Y 36.85, Z 0.00, A 0, B 0, C 0} C_DIS
LIN {X 193.25, Y 36.86, Z 0.00, A 0, B 0, C 0} C_DIS
LIN {X 193.03, Y 36.87, Z 0.00, A 0, B 0, C 0} C_DIS
LIN {X 192.81, Y 36.87, Z 0.00, A 0, B 0, C 0} C_DIS
LIN {X 192.60, Y 36.83, Z 0.00, A 0, B 0, C 0} C_DIS
LIN {X 192.38, Y 36.78, Z 0.00, A 0, B 0, C 0} C_DIS
LIN {X 192.17, Y 36.71, Z 0.00, A 0, B 0, C 0} C_DIS
LIN {X 191.96, Y 36.63, Z 0.00, A 0, B 0, C 0} C_DIS
LIN {X 191.75, Y 36.54, Z 0.00, A 0, B 0, C 0} C_DIS
LIN {X 191.54, Y 36.45, Z 0.00, A 0, B 0, C 0} C_DIS
LIN {X 191.33, Y 36.38, Z 0.00, A 0, B 0, C 0} C_DIS
LIN {X 191.11, Y 36.31, Z 0.00, A 0, B 0, C 0} C_DIS
LIN {X 190.90, Y 36.25, Z 0.00, A 0, B 0, C 0} C_DIS
LIN {X 190.69, Y 36.21, Z 0.00, A 0, B 0, C 0} C_DIS
LIN {X 190.47, Y 36.18, Z 0.00, A 0, B 0, C 0} C_DIS
LIN {X 190.25, Y 36.13, Z 0.00, A 0, B 0, C 0} C_DIS
LIN {X 190.04, Y 36.07, Z 0.00, A 0, B 0, C 0} C_DIS
LIN {X 189.83, Y 35.99, Z 0.00, A 0, B 0, C 0} C_DIS
LIN {X 189.62, Y 35.91, Z 0.00, A 0, B 0, C 0} C_DIS
LIN {X 189.41, Y 35.82, Z 0.00, A 0, B 0, C 0} C_DIS
LIN {X 189.20, Y 35.74, Z 0.00, A 0, B 0, C 0} C_DIS
LIN {X 188.99, Y 35.66, Z 0.00, A 0, B 0, C 0} C_DIS
LIN {X 188.78, Y 35.58, Z 0.00, A 0, B 0, C 0} C_DIS
LIN {X 188.57, Y 35.50, Z 0.00, A 0, B 0, C 0} C_DIS
LIN {X 188.35, Y 35.43, Z 0.00, A 0, B 0, C 0} C_DIS
LIN {X 188.14, Y 35.35, Z 0.00, A 0, B 0, C 0} C_DIS
LIN {X 187.93, Y 35.28, Z 0.00, A 0, B 0, C 0} C_DIS
LIN {X 187.72, Y 35.19, Z 0.00, A 0, B 0, C 0} C_DIS
LIN {X 187.51, Y 35.10, Z 0.00, A 0, B 0, C 0} C_DIS
LIN {X 187.31, Y 34.99, Z 0.00, A 0, B 0, C 0} C_DIS
LIN {X 187.11, Y 34.85, Z 0.00, A 0, B 0, C 0} C_DIS
LIN {X 186.91, Y 34.72, Z 0.00, A 0, B 0, C 0} C_DIS
LIN {X 186.70, Y 34.64, Z 0.00, A 0, B 0, C 0} C_DIS
LIN {X 186.49, Y 34.55, Z 0.00, A 0, B 0, C 0} C_DIS
LIN {X 186.29, Y 34.43, Z 0.00, A 0, B 0, C 0} C_DIS
LIN {X 186.11, Y 34.25, Z 0.00, A 0, B 0, C 0} C_DIS
LIN {X 185.92, Y 34.08, Z 0.00, A 0, B 0, C 0} C_DIS
LIN {X 185.72, Y 33.95, Z 0.00, A 0, B 0, C 0} C_DIS
LIN {X 185.51, Y 33.86, Z 0.00, A 0, B 0, C 0} C_DIS
LIN {X 185.30, Y 33.78, Z 0.00, A 0, B 0, C 0} C_DIS
LIN {X 185.10, Y 33.66, Z 0.00, A 0, B 0, C 0} C_DIS
LIN {X 184.90, Y 33.52, Z 0.00, A 0, B 0, C 0} C_DIS
LIN {X 184.70, Y 33.40, Z 0.00, A 0, B 0, C 0} C_DIS
LIN {X 184.49, Y 33.32, Z 0.00, A 0, B 0, C 0} C_DIS
LIN {X 184.28, Y 33.23, Z 0.00, A 0, B 0, C 0} C_DIS
LIN {X 184.08, Y 33.09, Z 0.00, A 0, B 0, C 0} C_DIS
LIN {X 183.90, Y 32.91, Z 0.00, A 0, B 0, C 0} C_DIS
LIN {X 183.71, Y 32.75, Z 0.00, A 0, B 0, C 0} C_DIS
LIN {X 183.51, Y 32.62, Z 0.00, A 0, B 0, C 0} C_DIS
LIN {X 183.31, Y 32.50, Z 0.00, A 0, B 0, C 0} C_DIS
LIN {X 183.12, Y 32.34, Z 0.00, A 0, B 0, C 0} C_DIS
LIN {X 182.94, Y 32.17, Z 0.00, A 0, B 0, C 0} C_DIS
LIN {X 182.74, Y 32.03, Z 0.00, A 0, B 0, C 0} C_DIS
LIN {X 182.54, Y 31.90, Z 0.00, A 0, B 0, C 0} C_DIS
LIN {X 182.34, Y 31.77, Z 0.00, A 0, B 0, C 0} C_DIS
LIN {X 182.16, Y 31.60, Z 0.00, A 0, B 0, C 0} C_DIS
LIN {X 181.97, Y 31.44, Z 0.00, A 0, B 0, C 0} C_DIS
LIN {X 181.77, Y 31.30, Z 0.00, A 0, B 0, C 0} C_DIS
LIN {X 181.57, Y 31.17, Z 0.00, A 0, B 0, C 0} C_DIS
LIN {X 181.38, Y 31.02, Z 0.00, A 0, B 0, C 0} C_DIS
LIN {X 181.19, Y 30.86, Z 0.00, A 0, B 0, C 0} C_DIS
LIN {X 181.01, Y 30.68, Z 0.00, A 0, B 0, C 0} C_DIS
LIN {X 180.83, Y 30.49, Z 0.00, A 0, B 0, C 0} C_DIS
LIN {X 180.65, Y 30.30, Z 0.00, A 0, B 0, C 0} C_DIS
LIN {X 180.48, Y 30.11, Z 0.00, A 0, B 0, C 0} C_DIS
LIN {X 180.30, Y 29.92, Z 0.00, A 0, B 0, C 0} C_DIS
LIN {X 180.11, Y 29.75, Z 0.00, A 0, B 0, C 0} C_DIS
LIN {X 179.93, Y 29.58, Z 0.00, A 0, B 0, C 0} C_DIS
LIN {X 179.73, Y 29.44, Z 0.00, A 0, B 0, C 0} C_DIS
LIN {X 179.53, Y 29.31, Z 0.00, A 0, B 0, C 0} C_DIS
LIN {X 179.34, Y 29.16, Z 0.00, A 0, B 0, C 0} C_DIS
LIN {X 179.15, Y 29.00, Z 0.00, A 0, B 0, C 0} C_DIS
LIN {X 178.96, Y 28.84, Z 0.00, A 0, B 0, C 0} C_DIS
LIN {X 178.78, Y 28.66, Z 0.00, A 0, B 0, C 0} C_DIS
LIN {X 178.61, Y 28.46, Z 0.00, A 0, B 0, C 0} C_DIS
LIN {X 178.44, Y 28.25, Z 0.00, A 0, B 0, C 0} C_DIS
LIN {X 178.28, Y 28.02, Z 0.00, A 0, B 0, C 0} C_DIS
LIN {X 178.13, Y 27.80, Z 0.00, A 0, B 0, C 0} C_DIS
